(* IEC 61131-3 sources: SmartHomeNew/ (part 3) *)

(* ---- GVL_POLICY.gvl ---- *)
VAR_GLOBAL
    // Policy bridges and centralized scenario ownership.
    G_Rule_Preheat_Request : BOOL := FALSE;
    G_Scenario_Request_Operator : E_SCENARIO_TYPE := E_SCENARIO_TYPE.SCENARIO_NONE;
    G_Scenario_Request_Gateway : E_SCENARIO_TYPE := E_SCENARIO_TYPE.SCENARIO_NONE;
    G_Scenario_Request_Rule : E_SCENARIO_TYPE := E_SCENARIO_TYPE.SCENARIO_NONE;
    G_Scenario_Intent : E_SCENARIO_TYPE := E_SCENARIO_TYPE.SCENARIO_NONE;
    G_Scenario_Source : E_SCENARIO_SOURCE := SRC_NONE;

    // Away-level policy state.
    // 0=none, 1=short, 2=medium, 3=long.
    G_Away_Active : BOOL := FALSE;
    G_Away_Level : BYTE := 0;
    G_Away_Start_MS : UDINT := 0;
    G_Away_Elapsed_MS : UDINT := 0;
    G_Away_Previous_Scenario : E_SCENARIO_TYPE := E_SCENARIO_TYPE.SCENARIO_PRESENCE;

    // Tuning defaults from ТЗ: short->medium after 2h, medium->long after 3d.
    G_Away_Short_To_Medium_MS : UDINT := 7200000;
    G_Away_Medium_To_Long_MS : UDINT := 259200000;

    G_Away_Simulation_Active : BOOL := FALSE;
    G_Away_Simulation_Intensity : REAL := 0.0;
    G_Away_Heating_Offset_C : REAL := 0.0;
    G_Away_Min_Heating_Setpoint_C : REAL := 15.0;
    G_Away_Long_Economy_Setpoint_C : REAL := 12.0;

    // Security alarm escalation policy.
    // On alarm: force long-away and publish a 5-minute lighting boost for
    // FB_Lighting_Blinds_Manager. This is a domain-level output override, not
    // a direct physical IO write.
    G_Security_Alarm_Force_Long_Away : BOOL := FALSE;
    G_Security_Alarm_Light_Boost_Active : BOOL := FALSE;
    G_Security_Alarm_Light_Boost_Start_MS : UDINT := 0;
    G_Security_Alarm_Light_Boost_Duration_MS : UDINT := 300000;

    // Entrance lighting assist policy.
    // Triggered by entrance door opening while dark. Darkness is configurable:
    // validated lux sensor below threshold and/or fallback to night flag.
    G_Entrance_Light_Assist_Active : BOOL := FALSE;
    G_Entrance_Light_Assist_Start_MS : UDINT := 0;
    G_Entrance_Light_Assist_Dark_Active : BOOL := FALSE;

    // Planned return / preheat policy.
    // Return time uses the current monotonic system-time domain. HMI/gateway may
    // set it as an absolute monotonic timestamp in the same domain.
    G_Away_Planned_Return_Enabled : BOOL := FALSE;
    G_Away_Planned_Return_MS : UDINT := 0;
    G_Away_Preheat_Lead_MS : UDINT := 10800000; // 3 hours
    G_Away_Return_Grace_MS : UDINT := 86400000; // 24 hours
    G_Away_Preheat_Target_C : REAL := 22.0;
    G_Away_Return_Preheat_Active : BOOL := FALSE;
    G_Away_Return_Grace_Active : BOOL := FALSE;
    G_Away_Return_Grace_Start_MS : UDINT := 0;
    G_Away_Return_Expired : BOOL := FALSE;

    // Restore state after short away. Downstream restore application is handled
    // by domain-specific code and should use this policy surface.
    G_Away_Restore_Requested : BOOL := FALSE;
    G_Away_Restore_Active : BOOL := FALSE;
    G_Away_Restore_Start_MS : UDINT := 0;
    G_Away_Restore_Duration_MS : UDINT := 60000;
    G_Away_Restore_Progress : REAL := 0.0;
END_VAR

(* ---- GVL_POWER_DOMAIN_SEGMENTATION_FABRIC.gvl ---- *)
VAR_GLOBAL
    Power_Domain_Segmentation_Valid : BOOL := FALSE;
    Power_Domain_Segmentation_Granted : BOOL := FALSE;

    Power_Domain_Boundaries_Canonical : BOOL := FALSE;
    Distributed_Power_Segmentation_Stable : BOOL := FALSE;
    Power_Reactivation_Isolation_Valid : BOOL := FALSE;

    Power_Segmentation_Causality_Valid : BOOL := FALSE;
    Power_Recovery_Ordering_Stable : BOOL := FALSE;

    Unsafe_Power_Resurrection_Detected : BOOL := FALSE;
    Partial_Power_Isolation_Asymmetry : BOOL := FALSE;
    Distributed_Power_Segmentation_Fork : BOOL := FALSE;

    Power_Domain_Segmentation_Epoch : UDINT := 0;
END_VAR

(* ---- GVL_Predictive_Diagnostics.gvl ---- *)
{attribute 'qualified_only'}
VAR_GLOBAL
    G_Diagnostics_State : ARRAY[1..64] OF ST_Predictive_Diagnostics_State;
END_VAR

VAR_GLOBAL RETAIN
    G_Total_Service_Recommendations : UDINT;
    G_Total_Urgent_Recommendations : UDINT;
END_VAR

VAR_GLOBAL
    G_Runtime_Valid : BOOL;
    G_Last_Update_MS : UDINT;

    G_Any_Degradation_Accumulating : BOOL;
    G_Any_Service_Recommended : BOOL;
    G_Any_Urgent_Service : BOOL;

    G_Status_Code : UINT;
    G_Status_Text : STRING(160);
END_VAR

(* ---- GVL_PRESENCE.gvl ---- *)
{attribute 'qualified_only'}
VAR_GLOBAL
    G_Any_Motion : BOOL := FALSE;
    G_Occupied : BOOL := TRUE;
    G_Auto_Away_Request : BOOL := FALSE;
    G_Last_Motion_TS : UDINT := 0;
END_VAR

(* ---- GVL_RECOVERY_GOVERNANCE.gvl ---- *)
VAR_GLOBAL
    // ======================================================
    // RECOVERY CLEANUP STATE
    // ======================================================
    // Centralized downstream recovery cleanup and residue state.
    // Recovery cleanup does not participate in upstream runtime
    // publication authority and must not feed back into runtime barrier.
    // ======================================================

    Recovery_Epoch : ULINT := 0;
    Recovery_Cleanup_Epoch : ULINT := 0;

    Recovery_Governance_Valid : BOOL := FALSE;
    Recovery_Cleanup_Completed : BOOL := FALSE;
    Recovery_Cleanup_Verified : BOOL := FALSE;

    Recovery_Quarantine_Active : BOOL := FALSE;
    Recovery_Forced_Safe_Mode : BOOL := FALSE;

    Recovery_Semantic_Residue_Detected : BOOL := FALSE;
    Recovery_Degraded_State_Residual : BOOL := FALSE;
    Recovery_Retained_State_Residual : BOOL := FALSE;

    Recovery_Last_Cleanup_Start_MS : UDINT := 0;
    Recovery_Last_Cleanup_End_MS : UDINT := 0;

    Recovery_Last_Error_Code : UDINT := 0;
    Recovery_Last_Error_Text : STRING(160) := '';

    Recovery_Invalidation_Count : UDINT := 0;
END_VAR

(* ---- GVL_Retain.gvl ---- *)
{attribute 'qualified_only'}
VAR_GLOBAL RETAIN
    G_Initialized : BOOL := FALSE; // Флаг инициализации retain-переменных

    // Compact RETAIN/NVRAM mirror for operational data only.
    // Logs, history, trends and blackbox archives must not consume RETAIN.
    G_NVRAM_Data : ARRAY[0..GVL_CONSTANTS.C_NVRAM_COMPACT_BYTES-1] OF BYTE;

    // Статистика котлов: оперативные счётчики наработки, нужны после рестарта.
    G_Boiler_Accumulated_MS : ARRAY[1..GVL_CONSTANTS.C_MAX_BOILERS] OF UDINT;
    G_Boiler_Work_Seconds : ARRAY[1..GVL_CONSTANTS.C_MAX_BOILERS] OF UDINT;

    // Результаты тестирования клапанов: компактное последнее состояние.
    G_Valve_Test_Results : ARRAY[1..GVL_CONSTANTS.C_MAX_MANIFOLDS] OF BOOL;

    // ПИН-коды доступа (храним хэши CRC32 для безопасности)
    // 16#9BE3E0A3 - это CRC32 от строки '1234'
    G_Access_Codes : ARRAY[1..GVL_CONSTANTS.C_MAX_ACCESS_CODES] OF DWORD := [16#9BE3E0A3, 16#4A89A12D, 16#F4DBDF21, 16#90F59C65, 16#0972D346, 0, 0, 0, 0, 0];

    // Зарегистрированные RFID/NFC метки (строковое представление UID)
    G_RFID_Tags : ARRAY[1..GVL_CONSTANTS.C_MAX_ACCESS_CODES] OF STRING(20) := ['A1B2C3D4', 'E5F67890', '', '', '', '', '', '', '', ''];
END_VAR

VAR_GLOBAL
    // Runtime blackbox buffer.
    // Kept in RAM only; CSV/file archive connection is a porting/module-stage task.
    G_BlackBox_Buffer : ARRAY[0..GVL_CONSTANTS.C_MAX_BLACKBOX_RECORDS-1] OF ST_BlackBox_Record;
    G_BlackBox_LastIndex : INT;
    G_BlackBox_Frozen : BOOL;

    // Presence playback history is non-safety behavioural data.
    // It is rebuilt during recording mode and must not consume RETAIN memory.
    G_Presence_History : ARRAY[0..GVL_CONSTANTS.C_MAX_PRESENCE_HISTORY-1] OF WORD;

    // Event history is an HMI/diagnostic runtime buffer.
    // It is repopulated by FB_History_Manager and must not consume RETAIN memory.
    G_History_Buffer : ARRAY[1..GVL_CONSTANTS.C_MAX_HISTORY_RECORDS] OF ST_History_Record;
    G_History_Write_Idx : INT := 1;
    G_History_Total_Events : UDINT;
END_VAR

(* ---- GVL_Runtime_Bus.gvl ---- *)
{attribute 'qualified_only'}
VAR_GLOBAL
    G_TX_Frames : ARRAY[1..128] OF ST_Runtime_Bus_Frame;
    G_RX_Frames : ARRAY[1..128] OF ST_Runtime_Bus_Frame;
END_VAR

VAR_GLOBAL RETAIN
    G_Last_Frame_Id : UDINT;
    G_Last_Sequence_Id : UDINT;
END_VAR

VAR_GLOBAL
    G_Runtime_Valid : BOOL;
    G_Last_Update_MS : UDINT;

    G_TX_Healthy : BOOL;
    G_RX_Healthy : BOOL;

    G_Any_Replication_Stale : BOOL;
    G_Any_Replication_Rejected : BOOL;

    G_Status_Code : UINT;
    G_Status_Text : STRING(160);
END_VAR

(* ---- GVL_Runtime_Discovery.gvl ---- *)
{attribute 'qualified_only'}
VAR_GLOBAL
    // Runtime discovery state is rebuilt by FB_Runtime_Node_Discovery
    // during cyclic execution. It must not consume RETAIN memory.
    G_Discovery_State : ARRAY[1..32] OF ST_Runtime_Node_Discovery_State;

    G_Runtime_Valid : BOOL;
    G_Last_Update_MS : UDINT;

    G_Any_Node_Quarantined : BOOL;
    G_Any_Discovery_Rejected : BOOL;

    G_Status_Code : UINT;
    G_Status_Text : STRING(160);
END_VAR

(* ---- GVL_RUNTIME_EPOCH.gvl ---- *)
VAR_GLOBAL
    // ======================================================
    // AUTHORITATIVE RUNTIME EPOCH STATE
    // ======================================================
    // Single authoritative runtime publication layer.
    // Used to stabilize scan-cycle visibility semantics.
    // ======================================================

    Runtime_Epoch : ULINT := 0;
    Runtime_Snapshot_Valid : BOOL := FALSE;
    Runtime_Snapshot_Published : BOOL := FALSE;
    Runtime_Runtime_Barrier_OK : BOOL := TRUE;
    Runtime_Impossible_State_Detected : BOOL := FALSE;

    Runtime_Last_Validation_Time_MS : UDINT := 0;
    Runtime_Last_Error_Code : UDINT := 0;
    Runtime_Last_Error_Text : STRING(160) := '';

    Runtime_Cycle_Start_MS : UDINT := 0;
    Runtime_Cycle_End_MS : UDINT := 0;

    Runtime_PLC_Authority_Valid : BOOL := FALSE;
    Runtime_IO_Publication_Allowed : BOOL := FALSE;

    Runtime_Barrier_Block_Count : UDINT := 0;
END_VAR

(* ---- GVL_Runtime_Restart_Continuity.gvl ---- *)
{attribute 'qualified_only'}
VAR_GLOBAL RETAIN
    G_Last_Stable_Config_Version : UDINT;
    G_Last_Known_Runtime_Healthy : BOOL;
    G_Last_Known_Quarantine_State : BOOL;

    G_Restore_Request : BOOL;
    G_Post_Restart_Validation_Request : BOOL;
END_VAR

VAR_GLOBAL
    G_Continuity_State : ST_Runtime_Restart_Continuity_State;

    G_Runtime_Valid : BOOL;
    G_Last_Update_MS : UDINT;

    G_Status_Code : UINT;
    G_Status_Text : STRING(160);
END_VAR

(* ---- GVL_RUNTIME_SCENARIO_VALIDATION.gvl ---- *)
{attribute 'qualified_only'}
VAR_GLOBAL
    // Runtime scenario validation. Observational only.
    // Validates that current safety/scenario context matches domain execution policy.

    G_Last_Update_MS : UDINT := 0;
    G_Validation_Executed : BOOL := FALSE;
    G_Validation_Valid : BOOL := TRUE;

    Idle_Context_Active : BOOL := FALSE;
    Security_Context_Active : BOOL := FALSE;
    Away_Context_Active : BOOL := FALSE;
    Presence_Context_Active : BOOL := FALSE;
    Fire_Context_Active : BOOL := FALSE;
    Gas_Context_Active : BOOL := FALSE;
    Leak_Context_Active : BOOL := FALSE;
    Global_Stop_Context_Active : BOOL := FALSE;
    Freeze_Context_Active : BOOL := FALSE;
    Heating_Demand_Context_Active : BOOL := FALSE;
    Vent_Boost_Context_Active : BOOL := FALSE;
    Access_Command_Context_Active : BOOL := FALSE;

    Idle_Context_Valid : BOOL := TRUE;
    Security_Context_Valid : BOOL := TRUE;
    Fire_Context_Valid : BOOL := TRUE;
    Gas_Context_Valid : BOOL := TRUE;
    Leak_Context_Valid : BOOL := TRUE;
    Global_Stop_Context_Valid : BOOL := TRUE;
    Freeze_Context_Valid : BOOL := TRUE;
    Heating_Context_Valid : BOOL := TRUE;
    Vent_Context_Valid : BOOL := TRUE;
    Access_Context_Valid : BOOL := TRUE;

    Any_Context_Invalid : BOOL := FALSE;
    Status_Code : UINT := 0;
    Status_Text : STRING(160) := '';
END_VAR

(* ---- GVL_Runtime_Sessions.gvl ---- *)
{attribute 'qualified_only'}
VAR_GLOBAL
    // Runtime session state is rebuilt by FB_Runtime_Session_Governance
    // during cyclic execution. It must not consume RETAIN memory.
    G_Local_Session : ST_Runtime_Node_Session;
    G_Remote_Sessions : ARRAY[1..16] OF ST_Runtime_Node_Session;

    G_Runtime_Valid : BOOL;
    G_Last_Update_MS : UDINT;

    G_Any_Stale_Session : BOOL;
    G_Any_Quarantined_Session : BOOL;

    G_Status_Code : UINT;
    G_Status_Text : STRING(160);
END_VAR

(* ---- GVL_RUNTIME_SNAPSHOT.gvl ---- *)
VAR_GLOBAL
    // ======================================================
    // IMMUTABLE RUNTIME SNAPSHOT AUTHORITY STATE
    // ======================================================
    // Centralized immutable publication snapshot governance.
    // Prevents mutable publication leakage across cycle boundaries.
    // ======================================================

    Snapshot_Epoch : ULINT := 0;
    Snapshot_Publication_Epoch : ULINT := 0;

    Snapshot_Frozen : BOOL := FALSE;
    Snapshot_Publication_Allowed : BOOL := FALSE;

    Snapshot_Copy_Valid : BOOL := FALSE;
    Snapshot_Isolation_Valid : BOOL := FALSE;
    Snapshot_Mutation_Detected : BOOL := FALSE;

    Snapshot_Runtime_Authority_Valid : BOOL := FALSE;
    Snapshot_Observability_Synchronized : BOOL := FALSE;

    Snapshot_Freeze_Start_MS : UDINT := 0;
    Snapshot_Last_Publication_MS : UDINT := 0;

    Snapshot_Last_Error_Code : UDINT := 0;
    Snapshot_Last_Error_Text : STRING(160) := '';

    Snapshot_Invalidation_Count : UDINT := 0;
END_VAR

(* ---- GVL_Safety_Bridge.gvl ---- *)
VAR_GLOBAL
    // === CO COMPARISON ===
    G_CO_Runtime : REAL;
    G_CO_Shadow  : REAL;
    G_CO_Diff    : REAL;

    // === METHANE COMPARISON ===
    G_Methane_Runtime : REAL;
    G_Methane_Shadow  : REAL;
    G_Methane_Diff    : REAL;

    // === SMOKE COMPARISON ===
    G_Smoke_Runtime : BOOL;
    G_Smoke_Shadow  : BOOL;
    G_Smoke_Diff    : BOOL;
END_VAR

(* ---- GVL_SAFETY_RECOVERY_CONFIG.gvl ---- *)
{attribute 'qualified_only'}
VAR_GLOBAL
    G_Stabilization_Delay_MS : UDINT := 5000;
    G_Stable_Time_Required_MS : UDINT := 3000;
    G_Cooldown_Time_MS : UDINT := 10000;
END_VAR

(* ---- GVL_Safety_Selector.gvl ---- *)
VAR_GLOBAL
    // === CONFIG SWITCHES ===
    G_Use_Shadow_CO : BOOL := FALSE;
    G_Use_Shadow_Methane : BOOL := FALSE;
    G_Use_Shadow_Smoke : BOOL := FALSE;

    // === EFFECTIVE SIGNALS ===
    G_CO_Effective : REAL;
    G_Methane_Effective : REAL;
    G_Smoke_Effective : BOOL;

    // === SHADOW QUALITY THRESHOLDS / POLICY ===
    G_CO_Shadow_Max_Diff : REAL := 5.0;
    G_Methane_Shadow_Max_Diff : REAL := 5.0;
    G_Block_Shadow_On_Mismatch : BOOL := TRUE;

    // === DEBOUNCE POLICY ===
    G_Shadow_Unstable_Cycles_Limit : INT := 5;

    // === RECOVERY POLICY (HYSTERESIS) ===
    G_CO_Shadow_Recovery_Diff : REAL := 2.0;
    G_Methane_Shadow_Recovery_Diff : REAL := 2.0;

    G_CO_Stable_Counter : INT := 0;
    G_Methane_Stable_Counter : INT := 0;
    G_Smoke_Stable_Counter : INT := 0;

    G_CO_Unstable_Counter : INT := 0;
    G_Methane_Unstable_Counter : INT := 0;
    G_Smoke_Unstable_Counter : INT := 0;

    // === EFFECTIVE ARRAYS FOR SAFETY FB ===
    G_CO_Effective_Array : ARRAY[1..GVL_CONSTANTS.C_MAX_CO_SENSORS] OF REAL;
    G_Methane_Effective_Array : ARRAY[1..GVL_CONSTANTS.C_MAX_METHANE_SENSORS] OF REAL;
    G_Smoke_Effective_Array : ARRAY[1..GVL_CONSTANTS.C_MAX_SMOKE_SENSORS] OF BOOL;
END_VAR

(* ---- GVL_SECURITY_ACCESS_INTENT.gvl ---- *)
{attribute 'qualified_only'}
VAR_GLOBAL
    G_Auto_Lock_Close_Request : BOOL := FALSE;
    G_Auto_Lock_Close_Accepted_By_Arbitration : BOOL := FALSE;
    G_Last_Auto_Lock_Request_MS : UDINT := 0;
    G_Status_Text : STRING(160) := 'Security access intent idle';
END_VAR

(* ---- GVL_SECURITY_WORKFLOW.gvl ---- *)
{attribute 'qualified_only'}
VAR_GLOBAL
    G_Arming_In_Progress : BOOL := FALSE;
    G_Arm_Delay_ET : TIME := T#0s;
    G_Arm_Delay_Q : BOOL := FALSE;

    G_Pin_Entry_Active : BOOL := FALSE;
    G_Entry_Delay_ET : TIME := T#0s;
    G_Entry_Delay_Q : BOOL := FALSE;
    G_Pin_Fail_Count : BYTE := 0;
    G_Max_Attempts : BYTE := 0;

    G_Disarm_Pending : BOOL := FALSE;
    G_2FA_Required : BOOL := FALSE;
    G_2FA_Send_Code_Req : BOOL := FALSE;

    G_Combined_Window_Active : BOOL := FALSE;
    G_Combined_Event_Count : INT := 0;
    G_Intrusion_Active_Count : INT := 0;
    G_Intrusion_Event_Count : INT := 0;

    G_Any_Sensor_Active : BOOL := FALSE;
    G_Door_Blocking_Open : BOOL := FALSE;
    G_Window_Blocking_Open : BOOL := FALSE;
    G_Status_Text : STRING(200) := '';
    G_Last_Update_MS : UDINT := 0;
END_VAR

(* ---- GVL_SEMANTIC_COMMIT.gvl ---- *)
VAR_GLOBAL
    // ======================================================
    // SEMANTIC PUBLICATION COMMIT STATE
    // ======================================================
    // Isolated semantic publication checkpoint coherence.
    // Downstream/publication continuity only.
    // Does not invalidate runtime barrier, PLC fencing,
    // immutable snapshots, distributed commit or IO authority.
    // ======================================================

    Semantic_Commit_Epoch : ULINT := 0;
    Semantic_Checkpoint_Epoch : ULINT := 0;
    Semantic_Publication_Commit_Epoch : ULINT := 0;

    Local_Semantic_Checkpoint_Epoch : ULINT := 0;
    Peer_Semantic_Checkpoint_Epoch : ULINT := 0;

    Local_Semantic_Commit_Epoch : ULINT := 0;
    Peer_Semantic_Commit_Epoch : ULINT := 0;

    Semantic_Checkpoint_Prepare_Active : BOOL := FALSE;
    Semantic_Checkpoint_Prepare_Valid : BOOL := FALSE;
    Semantic_Checkpoint_Ack_Valid : BOOL := FALSE;

    Semantic_Publication_Commit_Requested : BOOL := FALSE;
    Semantic_Publication_Commit_Confirmed : BOOL := FALSE;

    Semantic_Checkpoint_Mismatch : BOOL := FALSE;
    Semantic_Commit_Mismatch : BOOL := FALSE;
    Semantic_Rollback_Detected : BOOL := FALSE;
    Semantic_Replay_Fenced : BOOL := FALSE;
    Semantic_Checkpoint_Missing : BOOL := FALSE;

    // ======================================================
    // SEMANTIC COMMIT STABILIZATION FOUNDATION
    // ======================================================

    Semantic_Checkpoint_Drift_Suspected : BOOL := FALSE;
    Semantic_Checkpoint_Jitter_Suspected : BOOL := FALSE;
    Semantic_Commit_Replay_Storm_Suspected : BOOL := FALSE;

    Semantic_Commit_Stabilization_Required : BOOL := FALSE;
    Semantic_Commit_Stabilized : BOOL := FALSE;

    Semantic_Commit_Stabilization_Window_MS : UDINT := 3000;
    Semantic_Commit_Last_Stable_MS : UDINT := 0;

    // ======================================================
    // PASSIVE SEMANTIC TELEMETRY FOUNDATION
    // ======================================================

    Semantic_Drift_Event_Count : ULINT := 0;
    Semantic_Jitter_Event_Count : ULINT := 0;
    Semantic_Replay_Storm_Event_Count : ULINT := 0;

    Semantic_Last_Drift_MS : UDINT := 0;
    Semantic_Last_Jitter_MS : UDINT := 0;
    Semantic_Last_Replay_Storm_MS : UDINT := 0;

    Semantic_Stabilization_Telemetry_Valid : BOOL := FALSE;

    Semantic_Commit_Lease_Active : BOOL := FALSE;
    Semantic_Commit_Lease_Expired : BOOL := FALSE;
    Semantic_Commit_Timeout_MS : UDINT := 5000;

    Semantic_Commit_Last_Refresh_MS : UDINT := 0;
    Peer_Semantic_Commit_Last_Refresh_MS : UDINT := 0;

    Semantic_Commit_Valid : BOOL := FALSE;
    Semantic_Commit_Quarantine_Active : BOOL := FALSE;
    Semantic_Commit_Forced_Safe_Mode : BOOL := FALSE;

    Semantic_Commit_Last_Error_Code : UDINT := 0;
    Semantic_Commit_Last_Error_Text : STRING(160) := '';

    Semantic_Commit_Invalidation_Count : UDINT := 0;
END_VAR

(* ---- GVL_SEMANTIC_CONTINUITY.gvl ---- *)
VAR_GLOBAL
    // Global semantic continuity authority.
    Semantic_Continuity_Valid : BOOL := FALSE;
    Semantic_Continuity_Granted : BOOL := FALSE;
    Semantic_Continuity_Quarantine_Active : BOOL := TRUE;

    // Semantic authority proofs.
    Operator_Intent_Coherent : BOOL := FALSE;
    Policy_Intent_Coherent : BOOL := FALSE;
    Adaptive_Behavior_Coherent : BOOL := FALSE;
    Recovery_Intent_Coherent : BOOL := FALSE;
    Distributed_Semantic_Coherent : BOOL := FALSE;

    // Intent continuity.
    Declared_System_Intent_Valid : BOOL := FALSE;
    Runtime_Goal_Alignment_Valid : BOOL := FALSE;
    Optimization_Boundary_Valid : BOOL := FALSE;
    Autonomous_Adjustment_Valid : BOOL := FALSE;

    // Semantic drift detection.
    Goal_Drift_Detected : BOOL := FALSE;
    Policy_Divergence_Detected : BOOL := FALSE;
    Adaptive_Learning_Semantic_Skew : BOOL := FALSE;
    Recovery_Intent_Mismatch_Detected : BOOL := FALSE;
    Optimization_Authority_Corruption_Detected : BOOL := FALSE;
    Distributed_Semantic_Fragmentation_Detected : BOOL := FALSE;

    // Semantic epochs.
    Semantic_Continuity_Epoch : UDINT := 0;
    Semantic_Continuity_Epoch_Coherent : BOOL := FALSE;

    // Temporal semantic authority.
    Semantic_Last_Update_MS : UDINT := 0;
    Semantic_Lease_Expired : BOOL := TRUE;

    // Diagnostics.
    Semantic_Last_Error_Code : UDINT := 0;
    Semantic_Last_Error_Text : STRING(160) := '';
    Semantic_Invalidation_Count : UDINT := 0;
END_VAR

(* ---- GVL_SEMANTIC_DRIFT_OBSERVABILITY_FABRIC.gvl ---- *)
VAR_GLOBAL
    Semantic_Drift_Observability_Active : BOOL := TRUE;

    Semantic_Continuity_Observed : BOOL := FALSE;
    Semantic_Projection_Consistency_Observed : BOOL := FALSE;
    Distributed_Semantic_Alignment_Observed : BOOL := FALSE;

    Semantic_Drift_ReadOnly_Mode : BOOL := TRUE;
    Semantic_Drift_NoExecutionMutation : BOOL := TRUE;

    Semantic_Drift_Observed : BOOL := FALSE;
    Semantic_Lineage_Drift_Observed : BOOL := FALSE;
    Semantic_Projection_Decay_Observed : BOOL := FALSE;

    Semantic_Drift_Observation_Epoch : UDINT := 0;
END_VAR

(* ---- GVL_SEMANTIC_EPOCH_INVARIANCE_FABRIC.gvl ---- *)
VAR_GLOBAL
    // Deterministic semantic epoch invariance governance.
    Semantic_Epoch_Invariance_Valid : BOOL := FALSE;
    Semantic_Epoch_Invariance_Granted : BOOL := FALSE;
    Semantic_Epoch_Invariance_Quarantine_Active : BOOL := TRUE;

    // Cross-epoch semantic preservation proofs.
    Authority_Semantics_Invariant : BOOL := FALSE;
    CrossEpoch_Permission_Mapping_Stable : BOOL := FALSE;
    Semantic_Intent_Continuity_Valid : BOOL := FALSE;
    Governance_Meaning_Preservation_Coherent : BOOL := FALSE;
    Semantic_Evolution_Lineage_Traceable : BOOL := FALSE;

    // Semantic migration integrity.
    Explicit_Semantic_Migration_Governed : BOOL := FALSE;
    CrossEpoch_Semantic_Equivalence_Valid : BOOL := FALSE;
    Distributed_Semantic_Consensus_Stable : BOOL := FALSE;
    Semantic_Interpretation_Integrity_Valid : BOOL := FALSE;

    // Semantic epoch drift detectors.
    Semantic_Authority_Drift_Detected : BOOL := FALSE;
    CrossEpoch_Permission_Reinterpretation : BOOL := FALSE;
    Intent_To_Authority_Mismatch_Detected : BOOL := FALSE;
    Governance_Semantic_Fork_Detected : BOOL := FALSE;
    Semantic_Migration_Lineage_Gap_Detected : BOOL := FALSE;
    Distributed_Semantic_Divergence_Detected : BOOL := FALSE;

    // Semantic epochs.
    Semantic_Epoch_Invariance_Epoch : UDINT := 0;
    Semantic_Epoch_Invariance_Epoch_Coherent : BOOL := FALSE;

    // Temporal authority.
    Semantic_Epoch_Invariance_Last_Update_MS : UDINT := 0;
    Semantic_Epoch_Invariance_Lease_Expired : BOOL := TRUE;

    // Diagnostics.
    Semantic_Epoch_Invariance_Last_Error_Code : UDINT := 0;
    Semantic_Epoch_Invariance_Last_Error_Text : STRING(160) := '';
    Semantic_Epoch_Invariance_Invalidation_Count : UDINT := 0;
END_VAR

(* ---- GVL_SEMANTIC_PROGRESS.gvl ---- *)
VAR_GLOBAL
    // ======================================================
    // SEMANTIC PROGRESS CONTINUITY STATE
    // ======================================================
    // Isolated semantic execution continuity foundation.
    // Visibility/publication continuity only.
    // Does not invalidate runtime barrier,
    // PLC fencing, immutable snapshots or IO authority.
    // ======================================================

    Semantic_Progress_Epoch : ULINT := 0;
    Semantic_Continuity_Epoch : ULINT := 0;

    Semantic_Forward_Progress_Valid : BOOL := FALSE;
    Semantic_Execution_Continuity_OK : BOOL := FALSE;

    Semantic_Execution_Counter : ULINT := 0;
    Semantic_Last_Execution_Counter : ULINT := 0;

    Semantic_Progress_Last_Update_MS : UDINT := 0;
    Semantic_Progress_Timeout_MS : UDINT := 10000;

    Semantic_Stagnation_Detected : BOOL := FALSE;
    Semantic_Replay_Suspected : BOOL := FALSE;
    Semantic_Livelock_Suspected : BOOL := FALSE;
    Semantic_Deadlock_Suspected : BOOL := FALSE;

    Semantic_Progress_Lease_Active : BOOL := FALSE;
    Semantic_Progress_Lease_Expired : BOOL := FALSE;

    Semantic_Progress_Quarantine_Active : BOOL := FALSE;

    Semantic_Last_Error_Code : UDINT := 0;
    Semantic_Last_Error_Text : STRING(160) := '';

    Semantic_Invalidation_Count : UDINT := 0;
END_VAR

(* ---- GVL_Sensor_Shadow.gvl ---- *)
VAR_GLOBAL
    // === CO SHADOW PIPELINE EXPORT ===
    G_CO_Raw : REAL;
    G_CO_Processed : REAL;
    G_CO_Calibrated : REAL;
    G_CO_Error : BOOL;
    G_CO_Diag_Code : WORD;

    // === METHANE SHADOW PIPELINE EXPORT ===
    G_Methane_Raw : REAL;
    G_Methane_Processed : REAL;
    G_Methane_Calibrated : REAL;
    G_Methane_Error : BOOL;
    G_Methane_Diag_Code : WORD;

    // === SMOKE SHADOW PIPELINE EXPORT ===
    G_Smoke_Raw : BOOL;
    G_Smoke_Detected : BOOL;
END_VAR

(* ---- GVL_SIMULATION.gvl ---- *)
{attribute 'qualified_only'}
VAR_GLOBAL
    // ======================================================
    // ISOLATED SIMULATION / TEST REQUEST SURFACE
    // ======================================================
    // This GVL is a simulation/test request and status surface.
    // PRG_System_Simulation may write G_Test_* and G_Sim_* fields.
    //
    // Current runtime contract:
    // - simulation does NOT mutate production authority state;
    // - simulation does NOT write runtime/distributed/output GVLs;
    // - G_Sim_* fields are isolated effective test outputs;
    // - production consumers must not treat G_Sim_* as live sensor,
    //   command, fencing, transport or output authority without an
    //   explicit simulation injection boundary review.
    //
    // Note:
    // injection request flags are retained as test-control inputs.
    // A direct production injection bridge is not currently implemented.
    // ======================================================

    G_Simulation_Enable : BOOL := FALSE;

    // Scenario control
    G_Test_Scenario_ID : INT := 0; // 0=manual flags, 1=safety gas, 2=leak+low pressure, 3=sensor+predictive, 4=dual PLC, 5=full stress
    G_Test_Start : BOOL := FALSE;
    G_Test_Stop : BOOL := FALSE;
    G_Test_Scenario_Active : BOOL := FALSE;
    G_Test_Started_MS : UDINT := 0;
    G_Test_Duration_MS : UDINT := 30000;
    G_Test_Expected_Result_Code : INT := 0; // 0=none, 1=safety, 2=heating degraded, 3=role conflict, 4=full stress

    // Sensor fault injection requests
    G_Inject_Heating_Sensor_Fault : BOOL := FALSE;
    G_Inject_IO_Fault : BOOL := FALSE;
    G_Inject_Low_Pressure : BOOL := FALSE;
    G_Inject_Predictive_Pump_Fault : BOOL := FALSE;

    // Safety fault injection requests
    G_Inject_Gas_Alarm : BOOL := FALSE;
    G_Inject_Leak_Alarm : BOOL := FALSE;
    G_Inject_Smoke_Alarm : BOOL := FALSE;

    // PLC / role fault injection request
    G_Inject_Dual_PLC_Active : BOOL := FALSE;

    // Isolated effective simulation outputs. Production state is not overwritten by PRG_System_Simulation.
    G_Sim_Heating_Sensor_Fault : BOOL := FALSE;
    G_Sim_IO_Fault : BOOL := FALSE;
    G_Sim_Low_Pressure : BOOL := FALSE;
    G_Sim_Predictive_Pump_Fault : BOOL := FALSE;
    G_Sim_Gas_Alarm : BOOL := FALSE;
    G_Sim_Leak_Alarm : BOOL := FALSE;
    G_Sim_Smoke_Alarm : BOOL := FALSE;
    G_Sim_Dual_PLC_Active : BOOL := FALSE;

    // Test status
    G_Test_Running : BOOL := FALSE;
    G_Test_Result_OK : BOOL := FALSE;
    G_Test_Last_Result_Text : STRING(128) := 'No test executed';
END_VAR

(* ---- GVL_SMOKE_VERIFICATION.gvl ---- *)
{attribute 'qualified_only'}
VAR_GLOBAL
    G_Any_Smoke_Input_Active : BOOL;
    G_Smoke_Active_Count : UINT;
    G_Group_Active : ARRAY[1..3] OF BOOL;
    G_Group_Pair_Confirmed : ARRAY[1..3] OF BOOL;
    G_Group_Timer_Confirmed : ARRAY[1..3] OF BOOL;
    G_Verified_By_Pair : BOOL;
    G_Verified_By_Timer : BOOL;
    G_Verified_Group : INT := 0; // 1=basement, 2=floor1, 3=floor2
    G_Verified : BOOL;
    G_Status_Text : STRING(160) := 'Smoke verification idle';
    G_Last_Update_MS : UDINT := 0;
END_VAR

(* ---- GVL_STATE.gvl ---- *)
{attribute 'qualified_only'}
VAR_GLOBAL
    G_Floor_Temps : ARRAY[1..GVL_CONSTANTS.C_MAX_HEATING_CIRCUITS] OF REAL;
    G_Room_Temps : ARRAY[1..GVL_CONSTANTS.C_MAX_ZONES] OF REAL;
    G_Last_Valid_Room_Temps : ARRAY[1..GVL_CONSTANTS.C_MAX_ZONES] OF REAL;
    G_Last_Valid_Floor_Temps : ARRAY[1..GVL_CONSTANTS.C_MAX_HEATING_CIRCUITS] OF REAL;
    G_Temp_Sensor_Fault : ARRAY[1..GVL_CONSTANTS.C_MAX_ZONES] OF BOOL;
    G_Floor_Temp_Sensor_Fault : ARRAY[1..GVL_CONSTANTS.C_MAX_HEATING_CIRCUITS] OF BOOL;

    G_Flood_Warning : ARRAY[1..GVL_CONSTANTS.C_MAX_FLOOD_SENSORS] OF BOOL;
    G_Flood_Alarm : ARRAY[1..GVL_CONSTANTS.C_MAX_FLOOD_SENSORS] OF BOOL;
    G_Flood_Warning_Rise : ARRAY[1..GVL_CONSTANTS.C_MAX_FLOOD_SENSORS] OF BOOL;
    G_Flood_Alarm_Rise : ARRAY[1..GVL_CONSTANTS.C_MAX_FLOOD_SENSORS] OF BOOL;
    G_Flood_Alarm_Fall : ARRAY[1..GVL_CONSTANTS.C_MAX_FLOOD_SENSORS] OF BOOL;
END_VAR

(* ---- GVL_STATUS.gvl ---- *)
{attribute 'qualified_only'}
VAR_GLOBAL
    // ======================================================
    // MIXED GLOBAL STATUS SURFACE
    // ======================================================
    // Historical global status surface containing time, PLC role,
    // domain status, diagnostics and HMI text projections.
    //
    // Ownership boundaries:
    // - time fields are owned by PRG_Time_Service / monotonic time flow;
    // - PLC role fields are owned by PRG_PLC_Arbitration;
    // - domain status fields are projections owned by domain PRGs/FBs;
    // - diagnostics fields are diagnostics/status projections only;
    // - this GVL must not be used as a hidden distributed replication
    //   or direct-state HA apply surface.
    //
    // Note:
    // G_PLC_ID and G_Local_PLC_ID coexist as historical PLC ID surfaces.
    // Do not remove or merge without direct reference sweep.
    // ======================================================

    // Time / calendar status
    G_System_Time_MS : UDINT;
    G_Last_System_Time_MS : UDINT := 0;
    G_Time_Of_Day_MS : UDINT := 0;
    G_Current_Day : UINT := 1;
    G_Day_Of_Year : UINT := 1;
    G_Current_TOD : TOD;

    // Scenario / day-state status
    G_Current_Scenario : E_SCENARIO_TYPE := E_SCENARIO_TYPE.SCENARIO_NONE;
    G_Previous_Scenario : E_SCENARIO_TYPE := E_SCENARIO_TYPE.SCENARIO_NONE;
    G_Is_Night : BOOL;

    // PLC role / heartbeat authority projection.
    // Owner: PRG_PLC_Arbitration.
    G_PLC_ID : BYTE := 1;
    G_Is_Active_PLC : BOOL;
    G_Other_PLC_Is_Active : BOOL;

    G_Remote_PLC_Last_Seen_MS : UDINT;
    G_Remote_PLC_Alive : BOOL;

    G_Local_PLC_ID : BYTE := 1;
    G_Active_PLC_ID : BYTE := 1;
    G_Remote_PLC_Pulse : BOOL;

    // Domain / HMI status text projections
    G_Security_Status_Msg : STRING(200);
    G_Gas_Status_Msg : STRING(200);
    G_Flood_Status_Msg : STRING(200);
    G_Vent_Status_Msg : STRING(200);

    G_DHW_Status : ST_DHW_Status;
    G_Manifold_Status : ARRAY[1..GVL_CONSTANTS.C_MAX_MANIFOLDS] OF ST_Manifold_Status;
    G_Boiler_Status : ARRAY[1..GVL_CONSTANTS.C_MAX_BOILERS] OF ST_Boiler_Status;

    G_IO_Modules_Online : ARRAY[1..GVL_CONSTANTS.C_MAX_MODULES] OF BOOL;

    // Simulation / convenience status projections
    G_Sim_Active : BOOL;
    G_Wet_Zone_Light_Active : BOOL;

    // System mode / reason text projections
    G_System_Mode_Msg : STRING(200);
    G_System_Mode_Cause : STRING(200);
    G_System_Mode_Text : STRING(200);

    G_Evac_Target_Zone_Name : STRING(80);
    G_Evac_Hazard_Zone_Name : STRING(80);

    // Diagnostics projection surface
    G_Diagnostics : ST_System_Diagnostics;
    G_Diagnostics_Events : ARRAY[1..50] OF ST_Diagnostic_Event;
    G_Diagnostics_Count : INT := 0;
END_VAR

(* ---- GVL_SURVIVABILITY_INTELLIGENCE_FABRIC.gvl ---- *)
VAR_GLOBAL
    // Advisory/read-only survivability intelligence.
    Survivability_Intelligence_Active : BOOL := TRUE;
    Survivability_Intelligence_ReadOnly : BOOL := TRUE;
    Survivability_Intelligence_NoActuation : BOOL := TRUE;
    Survivability_Intelligence_NoAuthorityMutation : BOOL := TRUE;
    Survivability_Intelligence_NoRecoveryMutation : BOOL := TRUE;

    // Survivability continuum observations.
    System_Survivable : BOOL := FALSE;
    Degraded_But_Safe : BOOL := FALSE;
    Isolated_But_Stable : BOOL := FALSE;
    Partitioned_But_Survivable : BOOL := FALSE;
    Resource_Starved_But_Recoverable : BOOL := FALSE;

    // Essential function preservation advisories.
    Essential_Functions_Preserved : BOOL := FALSE;
    NonEssential_Shedding_Recommended : BOOL := FALSE;
    Telemetry_Rate_Reduction_Recommended : BOOL := FALSE;
    Heavy_Diagnostics_Defer_Recommended : BOOL := FALSE;
    Trend_Analytics_Defer_Recommended : BOOL := FALSE;
    Simulation_Defer_Recommended : BOOL := FALSE;

    // Long-duration degradation observations.
    LongDuration_Degradation_Observed : BOOL := FALSE;
    Chronic_Degradation_Risk_Increasing : BOOL := FALSE;
    Survivability_Pressure_Observed : BOOL := FALSE;
    Governance_Saturation_Pressure_Observed : BOOL := FALSE;
    Telemetry_Overload_Pressure_Observed : BOOL := FALSE;
    Distributed_Instability_Pressure_Observed : BOOL := FALSE;

    // Advisory diagnostics.
    Survivability_Advisory_Available : BOOL := FALSE;
    Survivability_Advisory_Code : STRING(255) := '';
    Survivability_Intelligence_Epoch : UDINT := 0;
END_VAR

(* ---- GVL_SYSTEM_COORDINATION.gvl ---- *)
{attribute 'qualified_only'}
VAR_GLOBAL
    G_System_Degraded : BOOL := FALSE;

    G_Block_Heating : BOOL := FALSE;
    G_Block_Ventilation : BOOL := FALSE;
    G_Block_Lighting_Override : BOOL := FALSE;
    G_Block_Sockets_Override : BOOL := FALSE;

    G_Coordination_Code : UDINT := 0;
END_VAR

(* ---- GVL_System_Diagnostics_Publication.gvl ---- *)
{attribute 'qualified_only'}
VAR_GLOBAL
    // Passive system diagnostics publication surface.
    // HMI/engineering diagnostics only: no command, output or runtime authority.
    G_System_Diagnostics : ST_System_Diagnostics;
    G_System_Diagnostics_Publication_Valid : BOOL := FALSE;
    G_System_Diagnostics_Status_Code : UINT := 0;
    G_System_Diagnostics_Status_Text : STRING(128) := 'System diagnostics publication inactive';
END_VAR

(* ---- GVL_TELEMETRY.gvl ---- *)
VAR_GLOBAL
    // Telemetry runtime authority.
    Telemetry_Runtime_Valid : BOOL := FALSE;
    Telemetry_Freshness_Valid : BOOL := FALSE;
    Telemetry_Lease_Expired : BOOL := TRUE;
    Telemetry_Quarantine_Active : BOOL := TRUE;

    // Command -> telemetry causality binding.
    Command_Telemetry_Causality_Valid : BOOL := FALSE;
    Command_Telemetry_Divergence_Detected : BOOL := TRUE;

    Command_Epoch : UDINT := 0;
    Telemetry_Epoch : UDINT := 0;
    Last_Acknowledged_Command_Epoch : UDINT := 0;

    // Physical actuator feedback authority.
    Actuator_Feedback_Valid : BOOL := FALSE;
    Actuator_Feedback_Fresh : BOOL := FALSE;
    Physical_Effect_Confirmed : BOOL := FALSE;
    Physical_Effect_Finalized : BOOL := FALSE;
    Physical_Target_Converged : BOOL := FALSE;
    Physical_Stable_Window_OK : BOOL := FALSE;
    Physical_Oscillation_Detected : BOOL := FALSE;
    Physical_Transition_Active : BOOL := FALSE;
    Physical_Convergence_Replay_Suspected : BOOL := FALSE;

    // Replay/staleness protection.
    Telemetry_Replay_Suspected : BOOL := FALSE;
    Last_Physical_Ack_Time_MS : UDINT := 0;
    Last_Physical_Convergence_MS : UDINT := 0;

    // Diagnostics.
    Telemetry_Last_Error_Code : UDINT := 0;
    Telemetry_Last_Error_Text : STRING(160) := '';
    Telemetry_Invalidation_Count : UDINT := 0;
END_VAR

(* ---- GVL_TEMPORAL_STABILITY.gvl ---- *)
VAR_GLOBAL
    // Global temporal stability authority.
    Temporal_Stability_Valid : BOOL := FALSE;
    Temporal_Stability_Granted : BOOL := FALSE;
    Temporal_Stability_Quarantine_Active : BOOL := TRUE;

    // Deterministic observation windows.
    Stability_Observation_Window_Active : BOOL := FALSE;
    Stability_Window_Start_MS : UDINT := 0;
    Stability_Window_Elapsed_MS : UDINT := 0;
    Stability_Window_Target_MS : UDINT := 5000;

    // Temporal convergence proofs.
    Post_Convergence_Stable : BOOL := FALSE;
    No_Oscillation_Detected : BOOL := FALSE;
    No_Relay_Chatter_Detected : BOOL := FALSE;
    Thermal_Slope_Stable : BOOL := FALSE;
    Pressure_Stable : BOOL := FALSE;
    Flow_Stable : BOOL := FALSE;

    // Delayed instability detection.
    Post_Convergence_Oscillation_Detected : BOOL := FALSE;
    Thermal_Inertia_Rebound_Detected : BOOL := FALSE;
    Pressure_Rebound_Detected : BOOL := FALSE;
    Relay_Chatter_Detected : BOOL := FALSE;
    Pump_Cavitation_Recovery_Detected : BOOL := FALSE;
    Delayed_Actuator_Divergence_Detected : BOOL := FALSE;

    // Temporal authority epochs.
    Temporal_Stability_Epoch : UDINT := 0;
    Temporal_Stability_Epoch_Coherent : BOOL := FALSE;

    // Temporal authority metadata.
    Temporal_Stability_Last_Update_MS : UDINT := 0;
    Temporal_Stability_Lease_Expired : BOOL := TRUE;

    // Diagnostics.
    Temporal_Stability_Last_Error_Code : UDINT := 0;
    Temporal_Stability_Last_Error_Text : STRING(160) := '';
    Temporal_Stability_Invalidation_Count : UDINT := 0;
END_VAR

(* ---- GVL_TEST.gvl ---- *)
{attribute 'qualified_only'}
VAR_GLOBAL
    G_Test_Enable : BOOL := FALSE;
    G_Test_Total_Checks : INT := 0;
    G_Test_Failed_Checks : INT := 0;
    G_Test_Passed : BOOL := TRUE;
    G_Test_Last_Failure_Index : INT := 0;
    G_Test_Last_Failure_Code : UDINT := 0;
    G_Test_Status_Msg : STRING(200) := 'Tests not run';

    // Runtime self-checks
    G_Ownership_Violation : BOOL := FALSE;
    G_Diagnostics_Duplicate_Event_Found : BOOL := FALSE;
    G_Diagnostics_Count_Out_Of_Range : BOOL := FALSE;
    G_Heating_Allocation_Budget_Exceeded : BOOL := FALSE;
    G_Heating_Allocation_Enabled_Not_Allowed : BOOL := FALSE;
    G_Safety_Latched_Without_Intent : BOOL := FALSE;

    // HP policy checks
    G_HP_Adjusted_Priority_Lower_Bound_Violation : BOOL := FALSE;
    G_HP_Adjusted_Allocation_Budget_Exceeded : BOOL := FALSE;
    G_HP_Adjusted_Allocation_Enabled_Not_Allowed : BOOL := FALSE;
    G_HP_Guest_Preheat_Config_Out_Of_Range : BOOL := FALSE;

    // Debug visibility
    G_HP_Manifold_Adjusted_Priority : ARRAY[1..GVL_CONSTANTS.C_MAX_MANIFOLDS] OF INT;
END_VAR

(* ---- GVL_TEST_INJECTION.gvl ---- *)
{attribute 'qualified_only'}
VAR_GLOBAL
    G_Inject_Enable : BOOL := FALSE;

    // Fault injection flags
    G_Inject_Gas_Level : REAL := 0.0;
    G_Inject_Force_Gas_Alarm_Reset : BOOL := FALSE;
    G_Inject_Force_IO_Offline : BOOL := FALSE;

    // Scenario runner
    G_Test_Step : INT := 0;
    G_Test_Timer_MS : UDINT := 0;
END_VAR

(* ---- GVL_TEST_PANEL.gvl ---- *)
{attribute 'qualified_only'}
VAR_GLOBAL
    // === CONTROL ===
    G_Enable : BOOL := FALSE;
    G_Scenario_ID : INT := 1;
    G_Scenario_ID_Prev : INT := 0;
    G_Scenario_Run : BOOL := FALSE;
    G_Scenario_Active : BOOL := FALSE;

    // === UI BLOCK: CURRENT TEST ===
    G_UI_00_Header : STRING(200) := '=== TEST PANEL ===';
    G_UI_01_Test : STRING(200) := 'Select G_Scenario_ID';
    G_UI_02_Change : STRING(200) := 'CHANGE: set scenario inputs';
    G_UI_03_Expected : STRING(200) := 'EXPECTED: see scenario instruction';
    G_UI_04_Result : STRING(200) := 'RESULT: Idle';
    G_UI_05_Error : STRING(200) := 'ERROR: -';
    G_UI_06_Actual : STRING(200) := 'ACTUAL: see numeric fields below';
    G_UI_07_Separator : STRING(200) := '----------------------------------------';

    // === UI BLOCK: NUMERIC FIELDS BELOW ===
    G_UI_10_Numeric_Block : STRING(200) := 'NUMERIC: Base / Expected / Actual / Delta';
    G_UI_11_Array_Block : STRING(200) := 'ARRAYS: Manifold expected / actual / enabled';
    G_UI_12_State_Block : STRING(200) := 'STATE: Safety / Block / Budget / Preheat';

    // === UX CONTROL ===
    G_Run_Counter : UDINT := 0;
    G_Last_Scenario_ID : INT := 0;
    G_Last_Result_Passed : BOOL := TRUE;
    G_Last_Fail_Code : UDINT := 0;
    G_Reset_Results_Request : BOOL := FALSE;
    G_Reset_Inputs_Request : BOOL := FALSE;
    G_Current_Test_Name : STRING(200) := '';
    G_Expected_Summary : STRING(200) := '';
    G_Actual_Summary : STRING(200) := '';
    G_Test_Result_Line : STRING(200) := 'Idle';
    G_Last_Result_Line : STRING(200) := '';
    G_Error_Text : STRING(200) := '';
    G_System_State_Line : STRING(200) := '';

    // === SCENARIO INPUTS ===
    G_Selected_Circuit : INT := 1;
    G_Input_Policy_Bias : INT := 0;
    G_Input_Guest_Preheat_Request : BOOL := FALSE;
    G_Input_Guest_Preheat_Enabled : BOOL := TRUE;
    G_Input_Guest_Preheat_Boost : INT := 2;
    G_Input_Max_Thermal_Budget : REAL := 2.0;
    G_Input_Block_Heating : BOOL := FALSE;
    G_Input_Safety_Stop : BOOL := FALSE;

    G_Input_Circuit_Enable : ARRAY[1..GVL_CONSTANTS.C_MAX_HEATING_CIRCUITS] OF BOOL;
    G_Input_Circuit_Bias : ARRAY[1..GVL_CONSTANTS.C_MAX_HEATING_CIRCUITS] OF INT;
    G_Input_Circuit_Guest_Preheat : ARRAY[1..GVL_CONSTANTS.C_MAX_HEATING_CIRCUITS] OF BOOL;

    G_Test_Description : STRING(200) := 'Idle';
    G_Test_What_To_Change : STRING(200) := '';
    G_Test_Expected_Text : STRING(200) := '';

    // === NUMERIC RESULT FIELDS ===
    G_Result_Mapped_Manifold : INT := 0;
    G_Result_Base_Priority : INT := 0;
    G_Result_Expected_Adjusted_Priority : INT := 0;
    G_Result_Actual_Adjusted_Priority : INT := 0;
    G_Result_Delta : INT := 0;

    G_Result_Manifold_Base_Priority : ARRAY[1..GVL_CONSTANTS.C_MAX_MANIFOLDS] OF INT;
    G_Result_Manifold_Expected_Priority : ARRAY[1..GVL_CONSTANTS.C_MAX_MANIFOLDS] OF INT;
    G_Result_Manifold_Actual_Priority : ARRAY[1..GVL_CONSTANTS.C_MAX_MANIFOLDS] OF INT;
    G_Result_Manifold_Delta : ARRAY[1..GVL_CONSTANTS.C_MAX_MANIFOLDS] OF INT;

    G_Result_Manifold_Allowed : ARRAY[1..GVL_CONSTANTS.C_MAX_MANIFOLDS] OF BOOL;
    G_Result_Manifold_Enabled : ARRAY[1..GVL_CONSTANTS.C_MAX_MANIFOLDS] OF BOOL;
    G_Result_Used_Thermal_Budget : REAL := 0.0;
    G_Result_Budget_Exceeded : BOOL := FALSE;

    G_Result_Passed : BOOL := TRUE;
    G_Result_Status_Msg : STRING(200) := 'Idle';
    G_Result_Fail_Code : UDINT := 0;
END_VAR

(* ---- GVL_TIME_MONOTONIC.gvl ---- *)
VAR_GLOBAL
    // ======================================================
    // MONOTONIC TIME GOVERNANCE STATE
    // ======================================================
    // Centralized monotonic authority layer.
    // Prevents rollback/reboot resurrection.
    // ======================================================

    Monotonic_Epoch : ULINT := 0;
    Boot_Generation_ID : ULINT := 0;

    Monotonic_Time_Valid : BOOL := FALSE;
    Monotonic_Time_Initialized : BOOL := FALSE;

    Startup_Quarantine_Active : BOOL := TRUE;
    Startup_Quarantine_Release_Allowed : BOOL := FALSE;
    Startup_Quarantine_Start_MS : UDINT := 0;
    Startup_Quarantine_Timeout_MS : UDINT := 10000;

    Time_Rollback_Detected : BOOL := FALSE;
    Retained_Time_Invalid : BOOL := FALSE;
    Time_Overflow_Detected : BOOL := FALSE;

    Last_Monotonic_Time_MS : UDINT := 0;
    Last_Validated_Time_MS : UDINT := 0;

    Monotonic_Last_Error_Code : UDINT := 0;
    Monotonic_Last_Error_Text : STRING(160) := '';

    Monotonic_Invalidation_Count : UDINT := 0;
END_VAR

(* ---- GVL_TIME_SERVICE.gvl ---- *)
{attribute 'qualified_only'}
VAR_GLOBAL
    // Published effective time for consumers
    G_Now_MS : UDINT;
    G_Time_Of_Day_MS : UDINT;
    G_Day_Of_Week : INT;
    G_Last_Now_MS : UDINT;
    G_Delta_MS : UDINT;
    G_Wrap_Detected : BOOL;

    // Simulation controls (HMI/runtime configurable)
    G_Sim_Enabled : BOOL;
    G_Sim_Frozen : BOOL;
    G_Sim_Time_Scale : REAL := 1.0;
    G_Sim_Now_MS : UDINT;
    G_Sim_Time_Of_Day_MS : UDINT;
    G_Sim_Day_Of_Week : INT := 1;
END_VAR

(* ---- GVL_TRANSPORT_FRESHNESS.gvl ---- *)
VAR_GLOBAL
    // ======================================================
    // TRANSPORT FRESHNESS GOVERNANCE STATE
    // ======================================================
    // Centralized transport freshness authority.
    // Prevents stale transport semantic publication.
    // ======================================================

    Transport_Epoch : ULINT := 0;
    Transport_Publication_Epoch : ULINT := 0;

    Transport_Freshness_Valid : BOOL := FALSE;
    Transport_Publication_Allowed : BOOL := FALSE;

    Transport_Lease_Valid : BOOL := FALSE;
    Transport_Lease_Expired : BOOL := FALSE;
    Transport_Lease_Timeout_MS : UDINT := 5000;

    Transport_Quarantine_Active : BOOL := FALSE;
    Transport_Reconnect_Stabilizing : BOOL := FALSE;

    Transport_Stale_Frame_Detected : BOOL := FALSE;
    Transport_Transaction_Mismatch : BOOL := FALSE;
    Transport_Snapshot_Invalid : BOOL := FALSE;

    Transport_Last_Refresh_MS : UDINT := 0;
    Transport_Last_Reconnect_MS : UDINT := 0;
    Transport_Last_Publication_MS : UDINT := 0;

    Transport_Last_Error_Code : UDINT := 0;
    Transport_Last_Error_Text : STRING(160) := '';

    Transport_Invalidation_Count : UDINT := 0;
END_VAR

(* ---- GVL_Trend.gvl ---- *)
VAR_GLOBAL
    // === TREND HMI DATA ===
    G_Trend_Avg : REAL;
    G_Trend_Min : REAL;
    G_Trend_Max : REAL;
    G_Trend_Up : BOOL;
    G_Trend_Down : BOOL;

    // === TREND BUFFER FOR HMI ===
    G_Trend_Buffer : ARRAY[1..50] OF REAL;
    G_Trend_Buffer_Index : INT;

    G_Trend_Buffer_Timestamps : ARRAY[1..50] OF UDINT;

    // === TREND META FOR HMI ===
    G_Trend_Valid_Count : INT;
    G_Trend_Is_Wrapped : BOOL;
    G_Trend_Last_Update_MS : UDINT;
    G_Trend_Param_Type : BYTE;

    // === MULTI-SIGNAL TREND FOUNDATION ===
    G_Trend_Selected_Channel : BYTE := 1;
    G_Trend_Channel2_Enabled : BOOL := FALSE;
    G_Trend_Buffer_2 : ARRAY[1..50] OF REAL;
    G_Trend_Buffer_2_Timestamps : ARRAY[1..50] OF UDINT;
    G_Trend_Buffer_2_Index : INT;
    G_Trend_Buffer_2_Valid_Count : INT;
    G_Trend_Buffer_2_Is_Wrapped : BOOL;
    G_Trend_Channel2_Param_Type : BYTE := 0;

    // === HMI-FACING TREND NORMALIZATION ===
    G_Trend_Active_Param_Type : BYTE;
    G_Trend_Active_Label : STRING(32);
    G_Trend_Channel1_Label : STRING(32) := 'Outdoor Temp';
    G_Trend_Channel2_Label : STRING(32) := 'Floor Temp';

    // === ACTIVE TREND VIEW FOR HMI ===
    G_Trend_Active_Value : REAL;
    G_Trend_Active_Timestamp : UDINT;
    G_Trend_Active_Index : INT;
    G_Trend_Active_Valid_Count : INT;
    G_Trend_Active_Is_Wrapped : BOOL;

END_VAR

(* ---- GVL_UNSAFE_TRANSITION_FORENSICS_FABRIC.gvl ---- *)
VAR_GLOBAL
    Unsafe_Transition_Forensics_Valid : BOOL := FALSE;
    Unsafe_Transition_Forensics_Granted : BOOL := FALSE;

    Unsafe_Transition_Lineage_Preserved : BOOL := FALSE;
    Forensic_Causality_Continuity_Valid : BOOL := FALSE;
    Distributed_Unsafe_Event_Consensus : BOOL := FALSE;

    Unsafe_Transition_Timeline_Stable : BOOL := FALSE;
    Historical_Safety_Lineage_Coherent : BOOL := FALSE;

    Unsafe_Transition_Hidden : BOOL := FALSE;
    Forensic_Lineage_Break_Detected : BOOL := FALSE;
    Historical_Safety_Gap_Detected : BOOL := FALSE;

    Unsafe_Transition_Forensics_Epoch : UDINT := 0;
END_VAR

(* ---- GVL_VENT_DOMAIN_STATUS.gvl ---- *)
{attribute 'qualified_only'}
VAR_GLOBAL
    // Ventilation domain status. Observational only.

    G_Runtime_Required : BOOL := FALSE;
    G_Runtime_Executed : BOOL := FALSE;
    G_Runtime_Idle_By_Design : BOOL := FALSE;
    G_Runtime_Blocked_By_Command : BOOL := FALSE;
    G_Emergency_Context_Active : BOOL := FALSE;
    G_Any_Supply_Fan_Active : BOOL := FALSE;
    G_Any_Exhaust_Fan_Active : BOOL := FALSE;
    G_Vent_Enable_Active : BOOL := FALSE;
    G_Last_Update_MS : UDINT := 0;
    G_Status_Code : UINT := 0;
    G_Status_Text : STRING(128) := '';
END_VAR

(* ---- GVL_VENT_OUTPUT.gvl ---- *)
VAR_GLOBAL
    // Ventilation output projection (decouples IO_Write from GVL_STATE)

    AO_Supply_Fans : ARRAY[1..GVL_CONSTANTS.C_MAX_SUPPLY_FANS] OF UINT;
    AO_Exhaust_Fans : ARRAY[1..GVL_CONSTANTS.C_MAX_EXHAUST_FANS] OF UINT;

    DO_Vent_Enable : BOOL := FALSE;
END_VAR

(* ---- GVL_WATER_EMERGENCY_OPEN.gvl ---- *)
{attribute 'qualified_only'}
VAR_GLOBAL
    // HMI/runtime surface for emergency temporary opening during active leak alarm.
    // Targets are four leak zones, not raw leak sensors:
    // 1 = зона 1 кухня (краны 1 ХВС + 2 ГВС),
    // 2 = зона 2 мастер-санузел (краны 3 ХВС + 4 ГВС),
    // 3 = зона 3 гостевые санузлы + постирочная (краны 5 ХВС + 6 ГВС),
    // 4 = зона 4 котельная / общий ввод (35 ХВС + 36 ГВС).
    G_Request_Open : BOOL := FALSE;
    G_Request_Close_Now : BOOL := FALSE;
    G_Target_Isolation_Group : INT := 0;
    G_Duration_Minutes : INT := 1; // allowed values: 1, 3, 5

    G_Open_Active : ARRAY[1..4] OF BOOL;
    G_Open_Start_MS : ARRAY[1..4] OF UDINT;
    G_Open_Duration_MS : ARRAY[1..4] OF UDINT;
    G_Open_Remaining_MS : ARRAY[1..4] OF UDINT;
    G_Open_Count_Today : ARRAY[1..4] OF INT;

    // Derived commands consumed by PRG_Water.
    // G_Open_Riser_* names are retained as legacy compatibility aliases for
    // leak zones 1..3; zone 4 uses common inlet 35/36.
    G_Open_Riser_1_Active : BOOL := FALSE;
    G_Open_Riser_2_Active : BOOL := FALSE;
    G_Open_Riser_3_Active : BOOL := FALSE;
    G_Open_Common_Inlet_Active : BOOL := FALSE;
    G_Any_Open_Active : BOOL := FALSE;

    G_Daily_Reset_MS : UDINT := 0;
    G_Last_Request_Accepted : BOOL := FALSE;
    G_Last_Request_Denied : BOOL := FALSE;
    G_Last_Denial_Code : UINT := 0;
    G_Last_Event_Group : INT := 0;
    G_Last_Event_MS : UDINT := 0;
    G_Status_Text : STRING(200) := '';
    G_Last_Update_MS : UDINT := 0;
END_VAR

(* ---- GVL_Water_Hydraulic_Graph.gvl ---- *)
{attribute 'qualified_only'}
VAR_GLOBAL
    G_Topology_Edge : ARRAY[1..64] OF ST_Water_Hydraulic_Topology_Edge;
    G_Isolation_Path : ARRAY[1..64] OF ST_Water_Isolation_Path_Runtime_State;

    G_Any_Shared_Trunk : BOOL;
    G_Any_Conflict : BOOL;
    G_Any_Global_Fallback_Required : BOOL;

    G_Runtime_Valid : BOOL;
    G_Last_Update_MS : UDINT;

    G_Status_Code : UINT;
    G_Status_Text : STRING(128);
END_VAR

(* ---- GVL_Water_Hydraulic_Topology.gvl ---- *)
{attribute 'qualified_only'}
VAR_GLOBAL
    G_Topology_Node : ARRAY[1..64] OF ST_Water_Hydraulic_Topology_Node;
    G_Isolation_Group : ARRAY[1..64] OF ST_Water_Hydraulic_Isolation_Group;

    G_Any_Ambiguous : BOOL;
    G_Any_Global_Fallback_Required : BOOL;

    G_Runtime_Valid : BOOL;
    G_Last_Update_MS : UDINT;

    G_Status_Code : UINT;
    G_Status_Text : STRING(128);
END_VAR

(* ---- GVL_Water_Isolation_Intent.gvl ---- *)
{attribute 'qualified_only'}
VAR_GLOBAL
    // ==============================================================================
    // Water/Flood isolation intent publication.
    // ==============================================================================
    //
    // Explicit authority augmentation layer.
    //
    // This layer publishes:
    // - selective isolation intent;
    // - per-zone close requests;
    // - fallback-to-global requirements.
    //
    // It does NOT directly own outputs.
    // Final authority remains inside runtime arbitration/safety layers.
    // ==============================================================================

    // Per-sensor / logical-zone isolation intent.
    G_Zone_Close_Requested : ARRAY[1..GVL_CONSTANTS.C_MAX_FLOOD_SENSORS] OF BOOL;

    // Valve-group visibility: 1..3 local risers, 4 common inlet 35/36.
    G_Valve_Group_Close_Requested : ARRAY[1..GVL_CONSTANTS.C_MAX_FLOOD_VALVES] OF BOOL;

    // Conservative fallback visibility.
    G_Global_Isolation_Requested : BOOL;

    // Explainability.
    G_Intent_Valid : BOOL;
    G_Status_Code : UINT;
    G_Status_Text : STRING(128);
END_VAR

(* ---- GVL_Water_Isolation_Runtime.gvl ---- *)
{attribute 'qualified_only'}
VAR_GLOBAL
    // ==============================================================================
    // Water/Flood isolation semantic publication surface.
    // ==============================================================================
    //
    // Observe/publish-first isolation governance.
    //
    // This layer publishes:
    // - selective isolation intent;
    // - fallback-to-global semantics;
    // - topology visibility;
    // - explainability.
    //
    // It does NOT directly own valve outputs.
    // ==============================================================================

    G_Isolation_Runtime_State : ARRAY[1..GVL_CONSTANTS.C_MAX_FLOOD_SENSORS] OF ST_Water_Isolation_Runtime_State;

    // Aggregated visibility.
    G_Any_Isolation_Requested : BOOL;
    G_Any_Selective_Isolation : BOOL;
    G_Global_Fallback_Required : BOOL;

    // Projection lifecycle.
    G_Runtime_Valid : BOOL;
    G_Last_Update_MS : UDINT;

    // Explainability.
    G_Status_Code : UINT;
    G_Status_Text : STRING(128);
END_VAR

(* ---- GVL_Water_Leak_Explainability.gvl ---- *)
{attribute 'qualified_only'}
VAR_GLOBAL
    // ==============================================================================
    // Water/Flood explainability compatibility publication surface.
    // ==============================================================================
    //
    // Compatibility/HMI/diagnostic publication layer.
    //
    // This GVL mirrors canonical Water runtime projection semantics for:
    // - HMI visibility;
    // - diagnostics continuity;
    // - migration stability;
    // - explainability publication.
    //
    // This GVL is NOT:
    // - runtime authority;
    // - valve authority;
    // - canonical routing root;
    // - supervisory aggregation owner.
    // ==============================================================================

    G_Leak_Visible : ARRAY[1..GVL_CONSTANTS.C_MAX_FLOOD_SENSORS] OF BOOL;
    G_Warning_Visible : ARRAY[1..GVL_CONSTANTS.C_MAX_FLOOD_SENSORS] OF BOOL;

    G_Mapping_Valid : ARRAY[1..GVL_CONSTANTS.C_MAX_FLOOD_SENSORS] OF BOOL;
    G_Selectively_Isolatable : ARRAY[1..GVL_CONSTANTS.C_MAX_FLOOD_SENSORS] OF BOOL;
    G_Global_Fallback_Required : ARRAY[1..GVL_CONSTANTS.C_MAX_FLOOD_SENSORS] OF BOOL;

    G_Leak_Confidence : ARRAY[1..GVL_CONSTANTS.C_MAX_FLOOD_SENSORS] OF REAL;

    G_Valve_Group_Id : ARRAY[1..GVL_CONSTANTS.C_MAX_FLOOD_SENSORS] OF UINT;
    G_Hydraulic_Zone_Id : ARRAY[1..GVL_CONSTANTS.C_MAX_FLOOD_SENSORS] OF UINT;

    G_Reason_Code : ARRAY[1..GVL_CONSTANTS.C_MAX_FLOOD_SENSORS] OF UINT;
    G_Reason_Text : ARRAY[1..GVL_CONSTANTS.C_MAX_FLOOD_SENSORS] OF STRING(128);

    G_Warning_Started_Event : ARRAY[1..GVL_CONSTANTS.C_MAX_FLOOD_SENSORS] OF BOOL;
    G_Leak_Confirmed_Event : ARRAY[1..GVL_CONSTANTS.C_MAX_FLOOD_SENSORS] OF BOOL;
    G_Leak_Cleared_Event : ARRAY[1..GVL_CONSTANTS.C_MAX_FLOOD_SENSORS] OF BOOL;

    G_Explainability_Valid : BOOL;
    G_Explainability_Status_Code : UINT;
    G_Explainability_Status_Text : STRING(128);
END_VAR

(* ---- GVL_Water_Orchestration.gvl ---- *)
{attribute 'qualified_only'}
VAR_GLOBAL
    G_Traversal_State : ARRAY[1..64] OF ST_Water_Graph_Traversal_State;
    G_Orchestration_State : ARRAY[1..64] OF ST_Water_Orchestration_Runtime_State;

    G_Topology_Version : UDINT;
    G_Config_Runtime_Ready : BOOL;

    G_Any_Traversal_Conflict : BOOL;
    G_Any_Escalation_Required : BOOL;

    G_Runtime_Valid : BOOL;
    G_Last_Update_MS : UDINT;

    G_Status_Code : UINT;
    G_Status_Text : STRING(128);
END_VAR

(* ---- GVL_WATER_OUTPUT.gvl ---- *)
VAR_GLOBAL
    // Legacy/global inlet valves.
    // 35 = общий ввод ХВС, 36 = общий ввод ГВС.
    DO_Water_Valve_35_Close : BOOL := FALSE;
    DO_Water_Valve_36_Close : BOOL := FALSE;

    // Local riser motorized ball valves with end switches.
    // 1 = стояк 1 ХВС, 2 = стояк 1 ГВС,
    // 3 = стояк 2 ХВС, 4 = стояк 2 ГВС,
    // 5 = стояк 3 ХВС, 6 = стояк 3 ГВС.
    DO_Water_Local_Valve_Open : ARRAY[1..6] OF BOOL;
    DO_Water_Local_Valve_Close : ARRAY[1..6] OF BOOL;

    DO_Water_Zone_Enable : ARRAY[1..GVL_CONSTANTS.C_MAX_WATER_ZONES] OF BOOL;
END_VAR

(* ---- GVL_Water_Output_Projection.gvl ---- *)
{attribute 'qualified_only'}
VAR_GLOBAL
    // Deterministic water output projection publication.

    G_Output_Projection_State : ARRAY[1..64] OF ST_Water_Output_Projection_State;

    // Aggregated visibility.
    G_Any_Output_Projected : BOOL;
    G_Any_Projection_Denied : BOOL;
    G_Global_Fallback_Projecting : BOOL;

    // Runtime.
    G_Runtime_Valid : BOOL;
    G_Last_Update_MS : UDINT;

    // Explainability.
    G_Status_Code : UINT;
    G_Status_Text : STRING(128);
END_VAR

(* ---- GVL_Water_Physical_Runtime.gvl ---- *)
{attribute 'qualified_only'}
VAR_GLOBAL
    G_Convergence_State : ARRAY[1..64] OF ST_Water_Physical_Convergence_State;
    G_Actuator_Diagnostics : ARRAY[1..64] OF ST_Water_Actuator_Diagnostics_State;

    G_Any_Convergence_Degraded : BOOL;
    G_Any_Diagnostics_Degraded : BOOL;
    G_Any_Escalation_Required : BOOL;

    G_Runtime_Valid : BOOL;
    G_Last_Update_MS : UDINT;

    G_Status_Code : UINT;
    G_Status_Text : STRING(128);
END_VAR

(* ---- GVL_Water_Runtime_Hardening.gvl ---- *)
{attribute 'qualified_only'}
VAR_GLOBAL
    G_Recovery_FSM : ARRAY[1..64] OF ST_Water_Recovery_FSM_State;
    G_Event_Log : ARRAY[1..128] OF ST_Water_Event_Log_Record;

    G_Runtime_Quarantine_Active : BOOL;
    G_Service_Mode_Active : BOOL;
    G_Maintenance_Mode_Active : BOOL;

    G_Any_Rollback_Required : BOOL;
    G_Any_Escalation_Required : BOOL;

    G_Runtime_Valid : BOOL;
    G_Last_Update_MS : UDINT;

    G_Status_Code : UINT;
    G_Status_Text : STRING(128);
END_VAR

(* ---- GVL_Water_Runtime_Supervisory_Publication.gvl ---- *)
{attribute 'qualified_only'}
VAR_GLOBAL
    // Water/Flood passive supervisory publication.
    // Observe/publish-only. No runtime or valve authority.

    G_Supervisory_Valid : BOOL;
    G_Last_Update_MS : UDINT;

    // Aggregated domain state.
    G_Any_Leak_Active : BOOL;
    G_Any_Warning_Active : BOOL;
    G_Any_Degraded_Mapping : BOOL;
    G_Selective_Isolation_Available : BOOL;
    G_Global_Fallback_Active : BOOL;

    // Current runtime visibility.
    G_Active_Global_Close_Path : BOOL;
    G_Active_Safety_Latch : BOOL;

    // Topology anchors.
    G_Affected_Hydraulic_Zone : UINT;
    G_Affected_Valve_Group : UINT;

    // Explainability aggregation.
    G_Status_Code : UINT;
    G_Status_Text : STRING(128);
END_VAR

(* ---- GVL_Water_Topology_Config_Source.gvl ---- *)
{attribute 'qualified_only'}
VAR_GLOBAL
    G_Source_Record : ARRAY[1..64] OF ST_Water_Topology_Config_Record;
END_VAR

VAR_GLOBAL RETAIN
    G_Source_Version : UDINT;
    G_Source_Valid : BOOL;
    G_Source_Activated_MS : UDINT;
END_VAR

VAR_GLOBAL
    G_Source_Status_Code : UINT;
    G_Source_Status_Text : STRING(128);
END_VAR

(* ---- GVL_Water_Valve_Runtime.gvl ---- *)
{attribute 'qualified_only'}
VAR_GLOBAL
    // ==============================================================================
    // Water/Flood valve governance publication.
    // ==============================================================================
    //
    // Observe-first valve governance and confirmation visibility.
    //
    // This layer publishes:
    // - valve runtime semantics;
    // - authority visibility;
    // - confirmation semantics;
    // - degraded-state visibility.
    //
    // This layer does NOT directly own physical outputs.
    // ==============================================================================

    G_Valve_Runtime_State : ARRAY[1..64] OF ST_Water_Valve_Runtime_State;

    // Aggregated visibility.
    G_Any_Valve_Degraded : BOOL;
    G_Any_Feedback_Invalid : BOOL;
    G_Any_Unsafe_Reopen_Denied : BOOL;

    // Lifecycle.
    G_Runtime_Valid : BOOL;
    G_Last_Update_MS : UDINT;

    // Explainability.
    G_Status_Code : UINT;
    G_Status_Text : STRING(128);
END_VAR

(* ---- GVL_WATER_VALVE_SERVICE.gvl ---- *)
{attribute 'qualified_only'}
VAR_GLOBAL
    G_Reset_Open_Block_Request : ARRAY[1..8] OF BOOL;
    G_Reset_All_Open_Blocks_Request : BOOL := FALSE;
    G_Reset_Confirm : BOOL := FALSE;

    G_Last_Reset_Accepted : BOOL := FALSE;
    G_Last_Reset_Denied : BOOL := FALSE;
    G_Last_Reset_Denial_Code : UINT := 0;
    G_Last_Reset_Valve_Index : INT := 0;
    G_Last_Reset_MS : UDINT := 0;
    G_Status_Text : STRING(200) := '';
END_VAR

(* ---- IValveController.st ---- *)
INTERFACE IValveController
METHOD OpenValve : BOOL
VAR_INPUT
    VI_Operator_ID : STRING(10);
    VI_Force : BOOL;
END_VAR
END_METHOD

METHOD CloseValve : BOOL
VAR_INPUT
    VI_Operator_ID : STRING(10);
    VI_Force : BOOL;
END_VAR
END_METHOD

METHOD GetStatus : BYTE
END_METHOD

(* ---- F_Modbus_RTU_CRC16.st ---- *)
FUNCTION F_Modbus_RTU_CRC16 : WORD
VAR_INPUT
    VI_Data : ARRAY[0..255] OF BYTE;
    VI_Length : UINT;
END_VAR

VAR
    L_CRC : WORD := 16#FFFF;
    L_i : UINT;
    L_j : INT;
    L_Temp : WORD;
END_VAR

// ======================================================
// MODBUS RTU CRC16
// ======================================================
// Standard Modbus RTU CRC16 implementation.
// Pure function without side effects.
// ======================================================

IF VI_Length = 0 THEN
    F_Modbus_RTU_CRC16 := 16#FFFF;
    RETURN;
END_IF;

FOR L_i := 0 TO (VI_Length - 1) DO

    L_CRC := L_CRC XOR BYTE_TO_WORD(VI_Data[L_i]);

    FOR L_j := 0 TO 7 DO

        L_Temp := L_CRC AND 16#0001;

        L_CRC := SHR(L_CRC, 1);

        IF L_Temp <> 0 THEN
            L_CRC := L_CRC XOR 16#A001;
        END_IF;

    END_FOR;

END_FOR;

F_Modbus_RTU_CRC16 := L_CRC;

END_FUNCTION

(* ---- IS_REAL_VALID.fun ---- *)
FUNCTION IS_REAL_VALID : BOOL
VAR_INPUT
    value : REAL;
END_VAR

// simple NaN / range guard
IS_REAL_VALID := (value > -1.0e6) AND (value < 1.0e6);

END_FUNCTION

(* ---- FB_ADS_Runtime_Adapter.st ---- *)
FUNCTION_BLOCK FB_ADS_Runtime_Adapter
VAR_INPUT
    VI_Enable : BOOL;
    VI_System_Time_MS : UDINT;
END_VAR
VAR
    L_Frame : ST_Runtime_Bus_Frame;
    L_TX_Index : UINT;
END_VAR

IF NOT VI_Enable THEN
    RETURN;
END_IF;

L_TX_Index := GVL_Runtime_Bus.G_Last_Sequence_Id;

IF (L_TX_Index >= 1)
   AND (L_TX_Index <= 128) THEN

    L_Frame := GVL_Runtime_Bus.G_TX_Frames[L_TX_Index];

    IF L_Frame.Frame_Valid THEN

        // ADS deterministic PLC-to-PLC runtime replication.
        // Transport adapter only confirms runtime-frame delivery eligibility.
        // It must never bypass distributed authority, sessions or safety barrier.
        IF GVL_Distributed_Authority.G_Distributed_Safety_Barrier_OK
           AND GVL_Runtime_Sessions.G_Runtime_Valid
           AND NOT GVL_Runtime_Sessions.G_Any_Stale_Session
           AND NOT GVL_Runtime_Sessions.G_Any_Quarantined_Session THEN

            L_Frame.Frame_Ack_Received := TRUE;
            L_Frame.Replication_Consistent := TRUE;
            L_Frame.Replication_Rejected := FALSE;

            L_Frame.Status_Code := 0;
            L_Frame.Status_Text :=
                'ADS runtime replication delivered';

        ELSE

            L_Frame.Frame_Ack_Received := FALSE;
            L_Frame.Replication_Consistent := FALSE;
            L_Frame.Replication_Rejected := TRUE;

            L_Frame.Status_Code := 2;
            L_Frame.Status_Text :=
                'ADS runtime replication blocked';

        END_IF;

        GVL_Runtime_Bus.G_TX_Frames[L_TX_Index] :=
            L_Frame;

        GVL_Runtime_Bus.G_TX_Healthy :=
            L_Frame.Replication_Consistent;

        GVL_Runtime_Bus.G_Any_Replication_Rejected :=
            L_Frame.Replication_Rejected;

    END_IF;

END_IF;

END_FUNCTION_BLOCK

(* ---- FB_Alarm_Compatibility_Package.st ---- *)
FUNCTION_BLOCK FB_Alarm_Compatibility_Package
VAR_INPUT
    VI_Alarm_Legacy : ST_Alarm_Record;
END_VAR
VAR_OUTPUT
    VO_OK : BOOL;
    VO_Alarm_Legacy_Roundtrip : ST_Alarm_Record;
END_VAR

VO_OK := TRUE;
VO_Alarm_Legacy_Roundtrip := VI_Alarm_Legacy;
END_FUNCTION_BLOCK

(* ---- FB_Alarm_Manager.st ---- *)
FUNCTION_BLOCK FB_Alarm_Manager
VAR_INPUT
    VI_System_Time_MS : UDINT; // Системное время (мс)
    VI_IsActivePLC : BOOL; // Флаг: Данный ПЛК является ведущим

    // Входы от подсистем
    VI_Gas_Alarm : BOOL; // Сигнал тревоги: Утечка газа
    VI_Fire_Alarm : BOOL; // Сигнал тревоги: Пожар
    VI_Flood_Alarm : BOOL; // Сигнал тревоги: Протечка воды
    VI_Security_Alarm : BOOL; // Сигнал тревоги: Охранная система
    VI_First_Fault_Active : BOOL; // Активна защёлкнутая первая причина деградации
    VI_First_Fault_Type : INT; // 1=IO,2=Sensor,3=Comm,4=Subsystem
    VI_First_Fault_Source : INT; // 1=Heating,2=DHW,3=Ventilation,4=Lighting,5=Access

    // Сообщения от подсистем (для детализации)
    VI_Security_Msg : STRING(200); // Детальное сообщение от охранной системы

    // Команды с HMI
    VI_Acknowledge_All : BOOL; // Команда: Квитировать все тревоги
    VI_Mute_Siren : BOOL; // Команда: Временное отключение сирены
END_VAR
VAR_IN_OUT
    VI_Boiler_Errors : ARRAY[1..GVL_CONSTANTS.C_MAX_BOILERS] OF BOOL; // Ошибки котлов
END_VAR
VAR_IN_OUT
    VIO_Next_Alarm_ID : UDINT; // Глобальный счетчик ID тревог
END_VAR
VAR_OUTPUT
    VO_Global_Critical : BOOL; // Есть неквитированные критические аварии
    VO_Global_Warning : BOOL;  // Есть неквитированные предупреждения
    VO_Siren_Active : BOOL;    // Требуется включение сирены
    VO_Active_Count : INT;     // Количество активных тревог
    VO_Unacked_Count : INT;    // Количество неквитированных тревог
    VO_Event_Pulse : BOOL;     // Пульс события для History bridge
    VO_Event_Code : UDINT;     // 1201=ack all, 1202=alarm cleared, 1203=alarm created
    VO_Event_Value : REAL;     // Доп. значение события

    VO_Alarm_List : ARRAY[1..GVL_CONSTANTS.C_MAX_ALARMS] OF ST_Alarm_Record; // Список активных тревог для HMI
END_VAR
VAR
    fbCompatAlarm : ARRAY[1..GVL_CONSTANTS.C_MAX_ALARMS] OF FB_Alarm_Compatibility_Package;
    L_i, L_j, L_k : INT;
    L_Target_Slot : INT;
    L_Min_Pri : INT;
    L_Pending_Alarms : ARRAY[1..10] OF ST_Alarm_Record;
    L_Pending_Count : INT := 0;

    // Фронты и антидребезг для детекции новых тревог
    T_Debounce_Gas : FB_System_Timer;
    T_Debounce_Fire : FB_System_Timer;
    T_Debounce_Flood : FB_System_Timer;
    T_Debounce_Security : FB_System_Timer;
    R_Trig_Gas : R_TRIG;
    R_Trig_Fire : R_TRIG;
    R_Trig_Flood : R_TRIG;
    R_Trig_Security : R_TRIG;
    R_Trig_First_Fault : R_TRIG;
    R_Trig_Boiler : ARRAY[1..GVL_CONSTANTS.C_MAX_BOILERS] OF R_TRIG;
    L_First_Fault_Source_Text : STRING(32);
    L_First_Fault_Type_Text : STRING(32);
    L_Event_Pulse_Latched : BOOL;
    L_Alarm_Compat_All_OK : BOOL;
    L_Alarm_First_Warning : STRING(255);
    L_Alarm_First_Warning_Latched : BOOL;
    L_Alarm_Shadow_Mismatch : BOOL;
    L_Alarm_Shadow_First_Mismatch : INT;
    L_Alarm_V2_Switch_Enabled : BOOL;
    L_Alarm_V2_Path_Ready : BOOL;
    L_Alarm_Using_Legacy_Fallback : BOOL;
    fbAlarmV2Core : FB_Alarm_V2_Core;
    fbHistoryV2Core : FB_History_V2_Core;
    fbBlackBoxV2Core : FB_BlackBox_V2_Core;
    L_BlackBox_V2_Snapshot_Shadow : ST_BlackBox_Snapshot_V2;
    L_History_V2_Shadow_Diff_Found : BOOL;
    L_History_V2_Shadow_First_Diff_Slot : INT;
    L_BlackBox_V2_Shadow_Diff_Found : BOOL;
    L_History_V2_Buffer_Shadow : ARRAY[1..GVL_CONSTANTS.C_MAX_HISTORY_RECORDS] OF ST_History_Event_V2;
    L_Alarm_V2_Shadow_Compare_Enabled : BOOL;
    L_Alarm_V2_Shadow_Diff_Found : BOOL;
    L_Alarm_V2_Shadow_First_Diff_Slot : INT;
    L_Alarm_V2_Event_Pulse : BOOL;
    L_Alarm_V2_Event_Code : UDINT;
    L_Alarm_V2_Event_Value : REAL;
    L_Alarm_V2_List_Shadow : ARRAY[1..GVL_CONSTANTS.C_MAX_ALARMS] OF ST_Alarm_Record;
    L_Alarm_V2_Next_ID_Shadow : UDINT;
END_VAR

VO_Event_Pulse := FALSE;
VO_Event_Code := 0;
VO_Event_Value := 0.0;

L_Alarm_Compat_All_OK := TRUE;
L_Alarm_First_Warning := '';
L_Alarm_First_Warning_Latched := FALSE;
L_Alarm_Shadow_Mismatch := FALSE;
L_Alarm_Shadow_First_Mismatch := 0;
L_Alarm_V2_Switch_Enabled := TRUE;
L_Alarm_V2_Path_Ready := FALSE;
L_Alarm_Using_Legacy_Fallback := TRUE;
L_Alarm_V2_Shadow_Compare_Enabled := TRUE;
L_Alarm_V2_Shadow_Diff_Found := FALSE;
L_Alarm_V2_Shadow_First_Diff_Slot := 0;
L_Alarm_V2_Event_Pulse := FALSE;
L_Alarm_V2_Event_Code := 0;
L_Alarm_V2_Event_Value := 0.0;
L_Alarm_V2_Next_ID_Shadow := VIO_Next_Alarm_ID;
L_History_V2_Shadow_Diff_Found := FALSE;
L_History_V2_Shadow_First_Diff_Slot := 0;
L_BlackBox_V2_Shadow_Diff_Found := FALSE;

// 1. Детекция новых тревог (антидребезг + передний фронт)
T_Debounce_Gas(IN := VI_Gas_Alarm, PT := T#100ms, VI_System_Time_MS := VI_System_Time_MS);
T_Debounce_Fire(IN := VI_Fire_Alarm, PT := T#100ms, VI_System_Time_MS := VI_System_Time_MS);
T_Debounce_Flood(IN := VI_Flood_Alarm, PT := T#500ms, VI_System_Time_MS := VI_System_Time_MS);
T_Debounce_Security(IN := VI_Security_Alarm, PT := T#100ms, VI_System_Time_MS := VI_System_Time_MS);

R_Trig_Gas(CLK := T_Debounce_Gas.Q);
R_Trig_Fire(CLK := T_Debounce_Fire.Q);
R_Trig_Flood(CLK := T_Debounce_Flood.Q);
R_Trig_Security(CLK := T_Debounce_Security.Q);
R_Trig_First_Fault(CLK := VI_First_Fault_Active);
FOR L_i := 1 TO GVL_CONSTANTS.C_MAX_BOILERS DO
    R_Trig_Boiler[L_i](CLK := VI_Boiler_Errors[L_i]);
END_FOR;

// 2. Добавление новых тревог в список (Кольцевой буфер)
L_Pending_Count := 0;
L_Event_Pulse_Latched := FALSE;

IF R_Trig_Gas.Q AND L_Pending_Count < 10 THEN
    L_Pending_Count := L_Pending_Count + 1;
    L_Pending_Alarms[L_Pending_Count].Timestamp_MS := VI_System_Time_MS;
    L_Pending_Alarms[L_Pending_Count].Source := 'Gas';
    L_Pending_Alarms[L_Pending_Count].Source_ID := 0;
    L_Pending_Alarms[L_Pending_Count].Message := 'Критическая концентрация газа!';
    L_Pending_Alarms[L_Pending_Count].Severity := E_ALERT_PRIORITY.ALERT_PRIORITY_CRITICAL;
    L_Pending_Alarms[L_Pending_Count].Is_Active := TRUE;
    L_Pending_Alarms[L_Pending_Count].Is_Acknowledged := FALSE;
END_IF;

IF R_Trig_Fire.Q AND L_Pending_Count < 10 THEN
    L_Pending_Count := L_Pending_Count + 1;
    L_Pending_Alarms[L_Pending_Count].Timestamp_MS := VI_System_Time_MS;
    L_Pending_Alarms[L_Pending_Count].Source := 'Fire';
    L_Pending_Alarms[L_Pending_Count].Source_ID := 0;
    L_Pending_Alarms[L_Pending_Count].Message := 'Обнаружено задымление!';
    L_Pending_Alarms[L_Pending_Count].Severity := E_ALERT_PRIORITY.ALERT_PRIORITY_CRITICAL;
    L_Pending_Alarms[L_Pending_Count].Is_Active := TRUE;
    L_Pending_Alarms[L_Pending_Count].Is_Acknowledged := FALSE;
END_IF;

IF R_Trig_Flood.Q AND L_Pending_Count < 10 THEN
    L_Pending_Count := L_Pending_Count + 1;
    L_Pending_Alarms[L_Pending_Count].Timestamp_MS := VI_System_Time_MS;
    L_Pending_Alarms[L_Pending_Count].Source := 'Flood';
    L_Pending_Alarms[L_Pending_Count].Source_ID := 0;
    L_Pending_Alarms[L_Pending_Count].Message := 'Обнаружена протечка воды!';
    L_Pending_Alarms[L_Pending_Count].Severity := E_ALERT_PRIORITY.ALERT_PRIORITY_CRITICAL;
    L_Pending_Alarms[L_Pending_Count].Is_Active := TRUE;
    L_Pending_Alarms[L_Pending_Count].Is_Acknowledged := FALSE;
END_IF;

IF R_Trig_Security.Q AND L_Pending_Count < 10 THEN
    L_Pending_Count := L_Pending_Count + 1;
    L_Pending_Alarms[L_Pending_Count].Timestamp_MS := VI_System_Time_MS;
    L_Pending_Alarms[L_Pending_Count].Source := 'Security';
    L_Pending_Alarms[L_Pending_Count].Source_ID := 0;
    L_Pending_Alarms[L_Pending_Count].Message := VI_Security_Msg;
    L_Pending_Alarms[L_Pending_Count].Severity := E_ALERT_PRIORITY.ALERT_PRIORITY_CRITICAL;
    L_Pending_Alarms[L_Pending_Count].Is_Active := TRUE;
    L_Pending_Alarms[L_Pending_Count].Is_Acknowledged := FALSE;
END_IF;

IF R_Trig_First_Fault.Q AND L_Pending_Count < 10 THEN
    L_Pending_Count := L_Pending_Count + 1;
    L_Pending_Alarms[L_Pending_Count].Timestamp_MS := VI_System_Time_MS;
    L_Pending_Alarms[L_Pending_Count].Source := 'Diagnostics';
    L_Pending_Alarms[L_Pending_Count].Source_ID := TO_BYTE(VI_First_Fault_Source);

    CASE VI_First_Fault_Type OF
        1: L_First_Fault_Type_Text := 'IO';
        2: L_First_Fault_Type_Text := 'Sensor';
        3: L_First_Fault_Type_Text := 'Comm';
        4: L_First_Fault_Type_Text := 'Subsystem';
        ELSE L_First_Fault_Type_Text := 'Unknown';
    END_CASE;

    CASE VI_First_Fault_Source OF
        1: L_First_Fault_Source_Text := 'Heating';
        2: L_First_Fault_Source_Text := 'DHW';
        3: L_First_Fault_Source_Text := 'Ventilation';
        4: L_First_Fault_Source_Text := 'Lighting';
        5: L_First_Fault_Source_Text := 'Access';
        ELSE L_First_Fault_Source_Text := 'Unknown';
    END_CASE;

    L_Pending_Alarms[L_Pending_Count].Message := CONCAT('Diagnostics root cause: ', CONCAT(L_First_Fault_Source_Text, CONCAT(' / ', L_First_Fault_Type_Text)));
    L_Pending_Alarms[L_Pending_Count].Severity := E_ALERT_PRIORITY.ALERT_PRIORITY_HIGH;
    L_Pending_Alarms[L_Pending_Count].Is_Active := TRUE;
    L_Pending_Alarms[L_Pending_Count].Is_Acknowledged := FALSE;
END_IF;

FOR L_j := 1 TO GVL_CONSTANTS.C_MAX_BOILERS DO
    IF R_Trig_Boiler[L_j].Q AND L_Pending_Count < 10 THEN
        L_Pending_Count := L_Pending_Count + 1;
        L_Pending_Alarms[L_Pending_Count].Timestamp_MS := VI_System_Time_MS;
        L_Pending_Alarms[L_Pending_Count].Source := 'Boiler';
        L_Pending_Alarms[L_Pending_Count].Source_ID := TO_BYTE(L_j);
        L_Pending_Alarms[L_Pending_Count].Message := CONCAT('Авария котла №', INT_TO_STRING(L_j));
        L_Pending_Alarms[L_Pending_Count].Severity := E_ALERT_PRIORITY.ALERT_PRIORITY_HIGH;
        L_Pending_Alarms[L_Pending_Count].Is_Active := TRUE;
        L_Pending_Alarms[L_Pending_Count].Is_Acknowledged := FALSE;
    END_IF;
END_FOR;

// Shadow comparison: execute Alarm V2 core on a separate shadow list.
// Legacy path remains authoritative; this is diagnostics only.
IF L_Alarm_V2_Shadow_Compare_Enabled THEN
    fbAlarmV2Core(
        VI_System_Time_MS := VI_System_Time_MS,
        VI_Pending_Alarms := L_Pending_Alarms,
        VIO_Alarm_List := L_Alarm_V2_List_Shadow,
        VIO_Next_Alarm_ID := L_Alarm_V2_Next_ID_Shadow,
        VO_Event_Pulse => L_Alarm_V2_Event_Pulse,
        VO_Event_Code => L_Alarm_V2_Event_Code,
        VO_Event_Value => L_Alarm_V2_Event_Value
    );
END_IF;

// Staging integration: Alarm V2 core is called behind the phase-4 switch scaffold.
// Current state: switch remains disabled, so legacy path stays authoritative.
IF L_Alarm_V2_Switch_Enabled AND L_Alarm_V2_Path_Ready THEN
    fbAlarmV2Core(
        VI_System_Time_MS := VI_System_Time_MS,
        VI_Pending_Alarms := L_Pending_Alarms,
        VIO_Alarm_List := VO_Alarm_List,
        VIO_Next_Alarm_ID := VIO_Next_Alarm_ID
    );
END_IF;

// Обработка очереди новых тревог с учетом приоритетов
FOR L_i := 1 TO L_Pending_Count DO
    fbCompatAlarm[L_i](VI_Alarm_Legacy := L_Pending_Alarms[L_i]);

    IF NOT fbCompatAlarm[L_i].VO_OK THEN
        L_Alarm_Compat_All_OK := FALSE;
    END_IF;

    IF (NOT L_Alarm_First_Warning_Latched) AND (NOT fbCompatAlarm[L_i].VO_OK) THEN
        L_Alarm_First_Warning := 'Translation issue';
        L_Alarm_First_Warning_Latched := TRUE;
    END_IF;

    IF fbCompatAlarm[L_i].VO_Alarm_Legacy_Roundtrip.ID <> L_Pending_Alarms[L_i].ID THEN
        L_Alarm_Shadow_Mismatch := TRUE;
        IF L_Alarm_Shadow_First_Mismatch = 0 THEN
            L_Alarm_Shadow_First_Mismatch := L_i;
        END_IF;
    END_IF;
    // Phase 4 scaffold: optional Alarm V2 switch point.
    // Current state: always remain on legacy behavior.
    // Future state: when Alarm V2 path is implemented and validated,
    // this block becomes the controlled branch point.
    IF L_Alarm_V2_Switch_Enabled AND L_Alarm_V2_Path_Ready THEN
        L_Alarm_Using_Legacy_Fallback := FALSE;
        // Guarded V2 pipeline is allowed by shadow validation.
        // Current runtime logic still keeps legacy action flow authoritative until next package.
    ELSE
        L_Alarm_Using_Legacy_Fallback := TRUE;
    END_IF;

    L_Target_Slot := 0;

    // 1. Ищем пустой слот
    FOR L_k := 1 TO GVL_CONSTANTS.C_MAX_ALARMS DO
        IF VO_Alarm_List[L_k].ID = 0 THEN
            L_Target_Slot := L_k;
            EXIT;
        END_IF;
    END_FOR;

    // 2. Ищем квитированную тревогу с наименьшим приоритетом
    IF L_Target_Slot = 0 THEN
        L_Min_Pri := 999;
        FOR L_k := 1 TO GVL_CONSTANTS.C_MAX_ALARMS DO
            IF VO_Alarm_List[L_k].Is_Acknowledged AND TO_INT(VO_Alarm_List[L_k].Severity) < L_Min_Pri THEN
                L_Min_Pri := TO_INT(VO_Alarm_List[L_k].Severity);
                L_Target_Slot := L_k;
            END_IF;
        END_FOR;
    END_IF;

    // 3. Ищем неквитированную тревогу с наименьшим приоритетом (если он ниже добавляемой)
    IF L_Target_Slot = 0 THEN
        L_Min_Pri := 999;
        FOR L_k := 1 TO GVL_CONSTANTS.C_MAX_ALARMS DO
            IF TO_INT(VO_Alarm_List[L_k].Severity) < L_Min_Pri AND TO_INT(VO_Alarm_List[L_k].Severity) < TO_INT(L_Pending_Alarms[L_i].Severity) THEN
                L_Min_Pri := TO_INT(VO_Alarm_List[L_k].Severity);
                L_Target_Slot := L_k;
            END_IF;
        END_FOR;
    END_IF;

    IF L_Target_Slot = 0 THEN
        // Буфер полон критических неквитированных тревог. Не затираем!
        CONTINUE;
    END_IF;

    VO_Alarm_List[L_Target_Slot] := L_Pending_Alarms[L_i];
    VO_Alarm_List[L_Target_Slot].ID := VIO_Next_Alarm_ID;
    VIO_Next_Alarm_ID := VIO_Next_Alarm_ID + 1;
    IF VIO_Next_Alarm_ID = 0 THEN VIO_Next_Alarm_ID := 1; END_IF;
    IF NOT L_Event_Pulse_Latched THEN
        VO_Event_Pulse := TRUE;
        VO_Event_Code := 1203;
        VO_Event_Value := TO_REAL(VO_Alarm_List[L_Target_Slot].Severity);
        L_Event_Pulse_Latched := TRUE;
    END_IF;
END_FOR;

// Shadow comparison results: compare legacy output and V2 shadow output.
IF L_Alarm_V2_Shadow_Compare_Enabled THEN
    FOR L_i := 1 TO GVL_CONSTANTS.C_MAX_ALARMS DO
        IF (VO_Alarm_List[L_i].ID <> L_Alarm_V2_List_Shadow[L_i].ID)
           OR (VO_Alarm_List[L_i].Is_Active <> L_Alarm_V2_List_Shadow[L_i].Is_Active)
           OR (VO_Alarm_List[L_i].Is_Acknowledged <> L_Alarm_V2_List_Shadow[L_i].Is_Acknowledged)
           OR (VO_Alarm_List[L_i].Severity <> L_Alarm_V2_List_Shadow[L_i].Severity) THEN
            L_Alarm_V2_Shadow_Diff_Found := TRUE;
            IF L_Alarm_V2_Shadow_First_Diff_Slot = 0 THEN
                L_Alarm_V2_Shadow_First_Diff_Slot := L_i;
            END_IF;
        END_IF;
    END_FOR;
END_IF;

// 3. Обновление статуса существующих тревог (ушли ли они?)
FOR L_i := 1 TO GVL_CONSTANTS.C_MAX_ALARMS DO
    IF VO_Alarm_List[L_i].ID <> 0 THEN
        IF VO_Alarm_List[L_i].Source = 'Gas' THEN VO_Alarm_List[L_i].Is_Active := VI_Gas_Alarm;
        ELSIF VO_Alarm_List[L_i].Source = 'Fire' THEN VO_Alarm_List[L_i].Is_Active := VI_Fire_Alarm;
        ELSIF VO_Alarm_List[L_i].Source = 'Flood' THEN VO_Alarm_List[L_i].Is_Active := VI_Flood_Alarm;
        ELSIF VO_Alarm_List[L_i].Source = 'Security' THEN VO_Alarm_List[L_i].Is_Active := VI_Security_Alarm;
        ELSIF VO_Alarm_List[L_i].Source = 'Diagnostics' THEN VO_Alarm_List[L_i].Is_Active := VI_First_Fault_Active;
        ELSIF VO_Alarm_List[L_i].Source = 'Boiler' THEN
            IF TO_INT(VO_Alarm_List[L_i].Source_ID) >= 1 AND TO_INT(VO_Alarm_List[L_i].Source_ID) <= GVL_CONSTANTS.C_MAX_BOILERS THEN
                VO_Alarm_List[L_i].Is_Active := VI_Boiler_Errors[TO_INT(VO_Alarm_List[L_i].Source_ID)];
            END_IF;
        END_IF;
    END_IF;
END_FOR;

// 4. Квитирование тревог
IF VI_Acknowledge_All THEN
    FOR L_i := 1 TO GVL_CONSTANTS.C_MAX_ALARMS DO
        IF VO_Alarm_List[L_i].ID <> 0 THEN
            VO_Alarm_List[L_i].Is_Acknowledged := TRUE;
        END_IF;
    END_FOR;

    IF NOT L_Event_Pulse_Latched THEN
        VO_Event_Pulse := TRUE;
        VO_Event_Code := 1201;
        VO_Event_Value := TO_REAL(VO_Unacked_Count);
        L_Event_Pulse_Latched := TRUE;
    END_IF;
END_IF;

// 4.5 Автоквитирование некритичных тревог, если они больше не активны
FOR L_i := 1 TO GVL_CONSTANTS.C_MAX_ALARMS DO
    IF VO_Alarm_List[L_i].ID <> 0 AND NOT VO_Alarm_List[L_i].Is_Active AND NOT VO_Alarm_List[L_i].Is_Acknowledged THEN
        IF VO_Alarm_List[L_i].Severity <> E_ALERT_PRIORITY.ALERT_PRIORITY_CRITICAL THEN
            VO_Alarm_List[L_i].Is_Acknowledged := TRUE;
        END_IF;
    END_IF;
END_FOR;

// 5. Очистка списка (удаление неактивных И квитированных тревог)
// В кольцевом буфере мы просто помечаем слот как пустой (ID = 0), без сдвига массива
FOR L_i := 1 TO GVL_CONSTANTS.C_MAX_ALARMS DO
    IF VO_Alarm_List[L_i].ID <> 0 AND NOT VO_Alarm_List[L_i].Is_Active AND VO_Alarm_List[L_i].Is_Acknowledged THEN
        // Удаляем тревогу
        VO_Alarm_List[L_i].ID := 0;
        IF NOT L_Event_Pulse_Latched THEN
            VO_Event_Pulse := TRUE;
            VO_Event_Code := 1202;
            VO_Event_Value := 0.0;
            L_Event_Pulse_Latched := TRUE;
        END_IF;
    END_IF;
END_FOR;

// Shadow bridge: Alarm -> History V2 (diagnostic only)
fbHistoryV2Core(
    VI_Event_Pulse := VO_Event_Pulse,
    VI_Event_Code := VO_Event_Code,
    VI_Event_Value := VO_Event_Value,
    VI_System_Time_MS := VI_System_Time_MS,
    VIO_History_Buffer := L_History_V2_Buffer_Shadow
);

// Shadow bridge: System -> BlackBox V2 (diagnostic only)
fbBlackBoxV2Core(
    VI_System_Time_MS := VI_System_Time_MS,
    VI_System_Mode := 0,
    VI_Critical_Alarm_Active := VO_Global_Critical,
    VI_Warning_Active := VO_Global_Warning,
    VI_First_Fault_Type := TO_BYTE(VI_First_Fault_Type),
    VI_First_Fault_Source := TO_BYTE(VI_First_Fault_Source),
    VI_Gas_Alarm := VI_Gas_Alarm,
    VI_Fire_Alarm := VI_Fire_Alarm,
    VI_Flood_Alarm := VI_Flood_Alarm,
    VO_Snapshot => L_BlackBox_V2_Snapshot_Shadow
);

// Shadow validation: History V2 / BlackBox V2
IF VO_Event_Pulse THEN
    IF (L_History_V2_Buffer_Shadow[1].Event_Code <> VO_Event_Code)
       OR (ABS(L_History_V2_Buffer_Shadow[1].Event_Value - VO_Event_Value) > 0.0001) THEN
        L_History_V2_Shadow_Diff_Found := TRUE;
        IF L_History_V2_Shadow_First_Diff_Slot = 0 THEN
            L_History_V2_Shadow_First_Diff_Slot := 1;
        END_IF;
    END_IF;
END_IF;

IF (L_BlackBox_V2_Snapshot_Shadow.Gas_Alarm <> VI_Gas_Alarm)
   OR (L_BlackBox_V2_Snapshot_Shadow.Fire_Alarm <> VI_Fire_Alarm)
   OR (L_BlackBox_V2_Snapshot_Shadow.Flood_Alarm <> VI_Flood_Alarm)
   OR (L_BlackBox_V2_Snapshot_Shadow.First_Fault_Type <> TO_BYTE(VI_First_Fault_Type))
   OR (L_BlackBox_V2_Snapshot_Shadow.First_Fault_Source <> TO_BYTE(VI_First_Fault_Source)) THEN
    L_BlackBox_V2_Shadow_Diff_Found := TRUE;
END_IF;

// Guarded V2 pipeline enable:
// V2 path is allowed only when no shadow diff is present in Alarm/History/BlackBox.
IF L_Alarm_V2_Switch_Enabled THEN
    IF (NOT L_Alarm_V2_Shadow_Diff_Found)
       AND (NOT L_History_V2_Shadow_Diff_Found)
       AND (NOT L_BlackBox_V2_Shadow_Diff_Found) THEN
        L_Alarm_V2_Path_Ready := TRUE;
        L_Alarm_Using_Legacy_Fallback := FALSE;
    ELSE
        L_Alarm_V2_Path_Ready := FALSE;
        L_Alarm_Using_Legacy_Fallback := TRUE;
    END_IF;
ELSE
    L_Alarm_V2_Path_Ready := FALSE;
    L_Alarm_Using_Legacy_Fallback := TRUE;
END_IF;

// 6. Подсчет статистики и формирование глобальных флагов
VO_Global_Critical := FALSE;
VO_Global_Warning := FALSE;
VO_Siren_Active := FALSE;
VO_Active_Count := 0;
VO_Unacked_Count := 0;

FOR L_i := 1 TO GVL_CONSTANTS.C_MAX_ALARMS DO
    IF VO_Alarm_List[L_i].ID <> 0 THEN
        IF VO_Alarm_List[L_i].Is_Active THEN
            VO_Active_Count := VO_Active_Count + 1;
        END_IF;

        IF NOT VO_Alarm_List[L_i].Is_Acknowledged THEN
            VO_Unacked_Count := VO_Unacked_Count + 1;

            IF VO_Alarm_List[L_i].Severity = E_ALERT_PRIORITY.ALERT_PRIORITY_CRITICAL THEN
                VO_Global_Critical := TRUE;
                // Сирена работает только для неквитированных критических тревог, если не включен Mute
                IF NOT VI_Mute_Siren THEN
                    VO_Siren_Active := TRUE;
                END_IF;
            ELSIF VO_Alarm_List[L_i].Severity = E_ALERT_PRIORITY.ALERT_PRIORITY_HIGH THEN
                VO_Global_Warning := TRUE;
            END_IF;
        END_IF;
    END_IF;
END_FOR;
// >>> BULK_SYNC_ANCHOR: FB_Alarm_Manager <<<

(* ---- FB_Astro_Timer.st ---- *)
FUNCTION_BLOCK FB_Astro_Timer
VAR_INPUT
    VI_System_Time_MS : UDINT;
    VI_Latitude : REAL := 55.75; // Москва (по умолчанию)
    VI_Longitude : REAL := 37.61;
    VI_Timezone : REAL := 3.0; // UTC+3
    VI_Day_Of_Year : UINT; // День года (1-365)
END_VAR
// >>> SYNC_TEST_MARKER_002 <<<
VAR_OUTPUT
    VO_Sunset_Time : TOD;
    VO_Sunrise_Time : TOD;
    VO_Is_Night : BOOL;
    VO_Current_TOD : TOD; // Текущее время суток
END_VAR
VAR
    L_Current_TOD : TOD;
    L_Pi : REAL := 3.14159265359;
    L_Rad : REAL := 3.14159265359 / 180.0;
    L_Deg : REAL := 180.0 / 3.14159265359;
    L_B : REAL;
    L_EoT : REAL;
    L_Declination : REAL;
    L_Cos_Omega : REAL;
    L_Omega : REAL;
    L_Sunrise_Local : REAL;
    L_Sunset_Local : REAL;
END_VAR

L_Current_TOD := GVL_STATUS.G_Current_TOD;
VO_Current_TOD := L_Current_TOD;

// Equation of Time (EoT) in minutes
L_B := 360.0 / 365.0 * TO_REAL(VI_Day_Of_Year - 81) * L_Rad;
L_EoT := 9.87 * SIN(2.0 * L_B) - 7.53 * COS(L_B) - 1.5 * SIN(L_B);

// Solar Declination in degrees
L_Declination := 23.45 * SIN(360.0 / 365.0 * TO_REAL(VI_Day_Of_Year + 284) * L_Rad);

// Hour angle
L_Cos_Omega := -TAN(VI_Latitude * L_Rad) * TAN(L_Declination * L_Rad);

IF L_Cos_Omega > 1.0 THEN
    L_Cos_Omega := 1.0; // Polar night
ELSIF L_Cos_Omega < -1.0 THEN
    L_Cos_Omega := -1.0; // Polar day
END_IF;

L_Omega := ACOS(L_Cos_Omega) * L_Deg;

// Sunrise and Sunset in local time (hours)
L_Sunrise_Local := 12.0 - (L_Omega / 15.0) - (L_EoT / 60.0) + (VI_Timezone * 15.0 - VI_Longitude) / 15.0;
L_Sunset_Local := 12.0 + (L_Omega / 15.0) - (L_EoT / 60.0) + (VI_Timezone * 15.0 - VI_Longitude) / 15.0;

// Handle bounds
IF L_Sunrise_Local < 0.0 THEN L_Sunrise_Local := L_Sunrise_Local + 24.0; END_IF;
IF L_Sunrise_Local >= 24.0 THEN L_Sunrise_Local := L_Sunrise_Local - 24.0; END_IF;
IF L_Sunset_Local < 0.0 THEN L_Sunset_Local := L_Sunset_Local + 24.0; END_IF;
IF L_Sunset_Local >= 24.0 THEN L_Sunset_Local := L_Sunset_Local - 24.0; END_IF;

// Конвертация в TOD
VO_Sunrise_Time := TO_TOD(TO_UDINT(L_Sunrise_Local * 3600000.0));
VO_Sunset_Time := TO_TOD(TO_UDINT(L_Sunset_Local * 3600000.0));

// ТЗ 15.2: Закат + 30 мин / Рассвет - 30 мин
VO_Is_Night := (L_Current_TOD > (VO_Sunset_Time + T#30m)) OR (L_Current_TOD < (VO_Sunrise_Time - T#30m));
// >>> SYNC_TEST_MARKER_FORCE <<<
// >>> BULK_SYNC_ANCHOR: FB_Astro_Timer <<<
END_FUNCTION_BLOCK

(* ---- FB_Behavior_Adapt.st ---- *)
FUNCTION_BLOCK FB_Behavior_Adapt
VAR_INPUT
    iScenario : E_System_Reason_Code;
    iSuccess : BOOL;
    iMeasuredValue : REAL;
    iZone : INT;
    iConfidence : REAL;
END_VAR

VAR
    L_Stats : ST_Scenario_Stats;
    L_Zone : ST_Zone_Adapt_State;
    L_Adjustment : REAL;
    L_Decay : REAL;
END_VAR

IF NOT GVL_BEHAVIOR_ADAPT.G_Adapt_Enabled THEN RETURN; END_IF;

// GLOBAL STATS
L_Stats := GVL_BEHAVIOR_ADAPT.G_Scenario_Stats[iScenario];
L_Stats.Activations := L_Stats.Activations + 1;

IF iSuccess THEN
    L_Stats.Success_Count := L_Stats.Success_Count + 1;
ELSE
    L_Stats.Failure_Count := L_Stats.Failure_Count + 1;
END_IF;

IF L_Stats.Activations > 0 THEN
    L_Stats.Success_Rate := REAL(L_Stats.Success_Count) / REAL(L_Stats.Activations);
END_IF;

// ZONE ADAPT WITH DECAY
IF (iScenario = REASON_SCENARIO_VENT_BOOST) AND (iZone >= 1) AND (iZone <= GVL_CONSTANTS.C_MAX_ZONES) THEN

    L_Zone := GVL_BEHAVIOR_ADAPT.G_VentBoost_Zone_Adapt[iZone];

    IF L_Zone.Zone_Weight = 0.0 THEN
        L_Zone.Zone_Weight := GVL_BEHAVIOR_ADAPT.G_Adapt_Default_Zone_Weight;
    END_IF;

    // DECAY
    L_Decay := GVL_BEHAVIOR_ADAPT.G_Decay_Factor;
    L_Zone.Zone_Weight := L_Zone.Zone_Weight * L_Decay;
    L_Zone.Confidence := L_Zone.Confidence * L_Decay;

    // STATS
    L_Zone.Activations := L_Zone.Activations + 1;

    IF iSuccess THEN
        L_Zone.Success_Count := L_Zone.Success_Count + 1;
    ELSE
        L_Zone.Failure_Count := L_Zone.Failure_Count + 1;
    END_IF;

    IF L_Zone.Activations > 0 THEN
        L_Zone.Success_Rate := REAL(L_Zone.Success_Count) / REAL(L_Zone.Activations);
    END_IF;

    // CONFIDENCE LEARNING
    IF iConfidence >= GVL_BEHAVIOR_ADAPT.G_Adapt_Min_Confidence THEN
        L_Zone.Confidence := L_Zone.Confidence +
            (iConfidence - L_Zone.Confidence) * GVL_BEHAVIOR_ADAPT.G_Confidence_Learning_Rate;
    END_IF;

    // UPDATE
    IF (L_Zone.Activations MOD GVL_BEHAVIOR_ADAPT.G_Adapt_Update_Threshold) = 0 THEN

        L_Adjustment :=
            (L_Zone.Success_Rate - 0.5)
            * GVL_BEHAVIOR_ADAPT.G_Adapt_Learning_Rate
            * L_Zone.Confidence;

        L_Zone.Zone_Weight := LIMIT(0.5, L_Zone.Zone_Weight + L_Adjustment, 2.0);

    END_IF;

    L_Zone.Last_Update_MS := GVL_TIME_SERVICE.G_Now_MS;

    GVL_BEHAVIOR_ADAPT.G_VentBoost_Zone_Adapt[iZone] := L_Zone;

END_IF;

GVL_BEHAVIOR_ADAPT.G_Scenario_Stats[iScenario] := L_Stats;
END_FUNCTION_BLOCK

(* ---- FB_BlackBox_Recorder.st ---- *)
FUNCTION_BLOCK FB_BlackBox_Recorder
VAR_INPUT
    VI_Current_Data : ST_BlackBox_Record;
    VI_Freeze       : BOOL;
END_VAR
VAR_OUTPUT
    VO_Frozen       : BOOL;
    VO_Records_Count: INT;
END_VAR
VAR
    L_Write_Index   : INT := 0;
    L_Initialized   : BOOL := FALSE;
END_VAR

IF NOT L_Initialized THEN
    L_Write_Index := GVL_Retain.G_BlackBox_LastIndex;
    IF L_Write_Index < 0 OR L_Write_Index >= GVL_CONSTANTS.C_MAX_BLACKBOX_RECORDS THEN
        L_Write_Index := 0;
        GVL_Retain.G_BlackBox_LastIndex := 0;
    END_IF;
    L_Initialized := TRUE;
END_IF;

IF VI_Freeze THEN
    GVL_Retain.G_BlackBox_Frozen := TRUE;
END_IF;

VO_Frozen := GVL_Retain.G_BlackBox_Frozen;

IF NOT GVL_Retain.G_BlackBox_Frozen THEN
    GVL_Retain.G_BlackBox_Buffer[L_Write_Index] := VI_Current_Data;
    GVL_Retain.G_BlackBox_LastIndex := L_Write_Index;

    L_Write_Index := L_Write_Index + 1;
    IF L_Write_Index >= GVL_CONSTANTS.C_MAX_BLACKBOX_RECORDS THEN
        L_Write_Index := 0;
    END_IF;
END_IF;

VO_Records_Count := GVL_CONSTANTS.C_MAX_BLACKBOX_RECORDS; // Размер кольцевого буфера
// >>> BULK_SYNC_ANCHOR: FB_BlackBox_Recorder <<<
END_FUNCTION_BLOCK

(* ---- FB_Blinds_V2_Staging.st ---- *)
FUNCTION_BLOCK FB_Blinds_V2_Staging
VAR_INPUT
    VI_Blind_ID : INT;
    VI_Enable : BOOL;
    VI_Position_Setpoint : BYTE;
    VI_Manual_Override : BOOL;
    VI_Scenario_ID : INT;
    VI_Safety_Mode : BOOL;
    VI_Position_Actual : BYTE;
    VI_Manual_Override_Active : BOOL;
    VI_Is_Moving : BOOL;
    VI_Alarm_Active : BOOL;
END_VAR
VAR_OUTPUT
    VO_Command_Shadow : ST_Blinds_Command_V2;
    VO_State_Shadow : ST_Blinds_State_V2;
END_VAR

VO_Command_Shadow.Position_Setpoint := VI_Position_Setpoint;
VO_State_Shadow.Position_Actual := VI_Position_Actual;
END_FUNCTION_BLOCK

(* ---- FB_Boiler_OpenTherm_Interface.st ---- *)
FUNCTION_BLOCK FB_Boiler_OpenTherm_Interface
VAR_INPUT
    VI_Enable : ARRAY[1..GVL_CONSTANTS.C_MAX_BOILERS] OF BOOL;
    VI_Setpoint : ARRAY[1..GVL_CONSTANTS.C_MAX_BOILERS] OF REAL;

    VI_OT_Online : ARRAY[1..GVL_CONSTANTS.C_MAX_BOILERS] OF BOOL;
    VI_OT_Error : ARRAY[1..GVL_CONSTANTS.C_MAX_BOILERS] OF BOOL;
END_VAR

VAR_OUTPUT
    VO_OT_Enable : ARRAY[1..GVL_CONSTANTS.C_MAX_BOILERS] OF BOOL;
    VO_OT_Setpoint : ARRAY[1..GVL_CONSTANTS.C_MAX_BOILERS] OF REAL;
    VO_OT_Command_Valid : ARRAY[1..GVL_CONSTANTS.C_MAX_BOILERS] OF BOOL;
END_VAR

VAR
    L_i : INT;
    L_Setpoint : REAL;
END_VAR

FOR L_i := 1 TO GVL_CONSTANTS.C_MAX_BOILERS DO

    VO_OT_Enable[L_i] := FALSE;
    VO_OT_Setpoint[L_i] := 0.0;
    VO_OT_Command_Valid[L_i] := FALSE;

    // ======================================================
    // DEFAULT SAFE COMMANDS
    // ======================================================
    GVL_OPENTHERM_ADAPTER.G_Cmd_Enable[L_i] := FALSE;
    GVL_OPENTHERM_ADAPTER.G_Cmd_Setpoint_x10[L_i] := 0;

    // ======================================================
    // COMMAND VALIDATION
    // ======================================================
    IF VI_Enable[L_i] AND VI_OT_Online[L_i] AND NOT VI_OT_Error[L_i] THEN

        L_Setpoint := LIMIT(20.0, VI_Setpoint[L_i], 80.0);

        // Publish logical command outputs
        VO_OT_Enable[L_i] := TRUE;
        VO_OT_Setpoint[L_i] := L_Setpoint;

        // Publish physical adapter commands
        GVL_OPENTHERM_ADAPTER.G_Cmd_Enable[L_i] := TRUE;
        GVL_OPENTHERM_ADAPTER.G_Cmd_Setpoint_x10[L_i] := REAL_TO_UINT(L_Setpoint * 10.0);

        // Command sequence tracking
        GVL_OPENTHERM_ADAPTER.G_Cmd_Seq[L_i] :=
            GVL_OPENTHERM_ADAPTER.G_Cmd_Seq[L_i] + 1;

        GVL_OPENTHERM_ADAPTER.G_Cmd_Last_Write_MS[L_i] :=
            GVL_STATUS.G_System_Time_MS;

        // Command valid only if adapter confirmed delivery
        VO_OT_Command_Valid[L_i] :=
            GVL_OPENTHERM_ADAPTER.G_Command_Ack[L_i] AND
            (NOT GVL_OPENTHERM_ADAPTER.G_Adapter_Error[L_i]) AND
            GVL_OPENTHERM_ADAPTER.G_Adapter_Online[L_i];

    END_IF;

END_FOR;

END_FUNCTION_BLOCK
